# B&R Automation Studio project AutomatedPongGame (part 4)

#### testSet_FieldControl_Idle.c
```c
/********************************************************************
 * COPYRIGHT - MyAutoMation-IT
 ********************************************************************
 * Author: Raivo Berends
 ********************************************************************/

#include <bur/plctypes.h>

#ifdef _DEFAULT_INCLUDES
#include <AsDefault.h>
#endif

#include "UnitTest.h"
#include "Library.h"
#include "CommonTypes.h"
#include <string.h>

_SETUP_TEST(void)
{
	FieldControlFB.FieldControl = &FieldControlStruct;
	FieldControlFB.FieldMotor = &FieldMotorStruct;
	FieldControlFB.InclinoSensor = &InclinoSensorStruct;

	memset(FieldControlFB.FieldControl, 0, sizeof(*FieldControlFB.FieldControl));
	memset(FieldControlFB.FieldMotor, 0, sizeof(*FieldControlFB.FieldMotor));
	memset(FieldControlFB.InclinoSensor, 0, sizeof(*FieldControlFB.InclinoSensor));

	FieldControlFB.FieldControl->STS.StateInt = STATE_IDLE;

	TEST_DONE;
}

_TEST Test_Idle_StaysIdle_WhenNotRunning(void)
{
	FieldControlFB.FieldControl->STS.Running = 0;

	FB_FieldControl(&FieldControlFB);

	TEST_ASSERT_EQUAL_INT(STATE_IDLE, FieldControlFB.FieldControl->STS.StateInt);

	TEST_DONE;
}

_TEST Test_Idle_TransitionsToRunning(void)
{
	FieldControlFB.FieldControl->STS.Running = 1;

	FB_FieldControl(&FieldControlFB);

	TEST_ASSERT_EQUAL_INT(STATE_RUNNING, FieldControlFB.FieldControl->STS.StateInt);

	TEST_DONE;
}

/*
B+R UnitTest: This is generated code.
Do not edit! Do not move!
Description: UnitTest Testprogramm infrastructure (TestSet).
LastUpdated: 2026-05-07 13:23:22Z
By B+R UnitTest Helper Version: 2.0.2.35
*/
UNITTEST_FIXTURES(fixtures)
{
	new_TestFixture("Test_Idle_StaysIdle_WhenNotRunning", Test_Idle_StaysIdle_WhenNotRunning),
	new_TestFixture("Test_Idle_TransitionsToRunning", Test_Idle_TransitionsToRunning),
};

UNITTEST_CALLER_COMPLETE_EXPLICIT(testSet_FieldControl_Idle, "testSet_FieldControl_Idle", setupTest, 0, fixtures, 0, 0, 0);
```

#### testSet_FieldControl_Running.c
```c
/********************************************************************
 * COPYRIGHT - MyAutoMation-IT
 ********************************************************************
 * Author: Raivo Berends
 ********************************************************************/

#include <bur/plctypes.h>

#ifdef _DEFAULT_INCLUDES
#include <AsDefault.h>
#endif

#include "UnitTest.h"
#include "Library.h"
#include "CommonTypes.h"
#include <string.h>

_SETUP_TEST(void)
{
	FieldControlFB.FieldControl = &FieldControlStruct;
	FieldControlFB.FieldMotor = &FieldMotorStruct;
	FieldControlFB.InclinoSensor = &InclinoSensorStruct;

	memset(FieldControlFB.FieldControl, 0, sizeof(*FieldControlFB.FieldControl));
	memset(FieldControlFB.FieldMotor, 0, sizeof(*FieldControlFB.FieldMotor));
	memset(FieldControlFB.InclinoSensor, 0, sizeof(*FieldControlFB.InclinoSensor));

	FieldControlFB.FieldControl->STS.StateInt = STATE_RUNNING;

	TEST_DONE;
}

_TEST Test_Running_ResetsStopCommand(void)
{
	FieldControlFB.FieldMotor->CS.Stop = 1;

	FB_FieldControl(&FieldControlFB);

	TEST_ASSERT_EQUAL_INT(0, FieldControlFB.FieldMotor->CS.Stop);

	TEST_DONE;
}

_TEST Test_Running_DisablesJogNeg_WhenAtMaxAngle(void)
{
	FieldControlFB.FieldControl->STS.CurrentAngle = MAX_ANGLE;

	FieldControlFB.FieldMotor->HMI.MoveJogNeg = 1;

	FB_FieldControl(&FieldControlFB);

	TEST_ASSERT_EQUAL_INT(0, FieldControlFB.FieldMotor->HMI.MoveJogNeg);

	TEST_DONE;
}

_TEST Test_Running_DisablesJogNeg_WhenAboveMaxAngle(void)
{
	FieldControlFB.FieldControl->STS.CurrentAngle = 25.0;

	FieldControlFB.FieldMotor->HMI.MoveJogNeg = 1;

	FB_FieldControl(&FieldControlFB);

	TEST_ASSERT_EQUAL_INT(0, FieldControlFB.FieldMotor->HMI.MoveJogNeg);

	TEST_DONE;
}

_TEST Test_Running_DisablesJogPos_WhenAtMinAngle(void)
{
	FieldControlFB.FieldControl->STS.CurrentAngle = MIN_ANGLE;

	FieldControlFB.FieldMotor->HMI.MoveJogPos = 1;

	FB_FieldControl(&FieldControlFB);

	TEST_ASSERT_EQUAL_INT(0, FieldControlFB.FieldMotor->HMI.MoveJogPos);

	TEST_DONE;
}

_TEST Test_Running_DisablesJogPos_WhenBelowMinAngle(void)
{
	FieldControlFB.FieldControl->STS.CurrentAngle = 0.0;

	FieldControlFB.FieldMotor->HMI.MoveJogPos = 1;

	FB_FieldControl(&FieldControlFB);

	TEST_ASSERT_EQUAL_INT(0, FieldControlFB.FieldMotor->HMI.MoveJogPos);

	TEST_DONE;
}

_TEST Test_Running_DoesNotChangeJogCommands_WithinLimits(void)
{
	FieldControlFB.FieldControl->STS.CurrentAngle = 10.0;

	FieldControlFB.FieldMotor->HMI.MoveJogNeg = 1;
	FieldControlFB.FieldMotor->HMI.MoveJogPos = 1;

	FB_FieldControl(&FieldControlFB);

	TEST_ASSERT_EQUAL_INT(1, FieldControlFB.FieldMotor->HMI.MoveJogNeg);
	TEST_ASSERT_EQUAL_INT(1, FieldControlFB.FieldMotor->HMI.MoveJogPos);

	TEST_DONE;
}

_TEST Test_Running_MaxAngle_DoesNotChangeJogPos(void)
{
	FieldControlFB.FieldControl->STS.CurrentAngle = MAX_ANGLE;

	FieldControlFB.FieldMotor->HMI.MoveJogNeg = 1;
	FieldControlFB.FieldMotor->HMI.MoveJogPos = 1;

	FB_FieldControl(&FieldControlFB);

	TEST_ASSERT_EQUAL_INT(0, FieldControlFB.FieldMotor->HMI.MoveJogNeg);
	TEST_ASSERT_EQUAL_INT(1, FieldControlFB.FieldMotor->HMI.MoveJogPos);

	TEST_DONE;
}
/*
B+R UnitTest: This is generated code.
Do not edit! Do not move!
Description: UnitTest Testprogramm infrastructure (TestSet).
LastUpdated: 2026-05-07 13:23:22Z
By B+R UnitTest Helper Version: 2.0.2.35
*/
UNITTEST_FIXTURES(fixtures)
{
	new_TestFixture("Test_Running_ResetsStopCommand", Test_Running_ResetsStopCommand),
	new_TestFixture("Test_Running_DisablesJogNeg_WhenAtMaxAngle", Test_Running_DisablesJogNeg_WhenAtMaxAngle),
	new_TestFixture("Test_Running_DisablesJogNeg_WhenAboveMaxAngle", Test_Running_DisablesJogNeg_WhenAboveMaxAngle),
	new_TestFixture("Test_Running_DisablesJogPos_WhenAtMinAngle", Test_Running_DisablesJogPos_WhenAtMinAngle),
	new_TestFixture("Test_Running_DisablesJogPos_WhenBelowMinAngle", Test_Running_DisablesJogPos_WhenBelowMinAngle),
	new_TestFixture("Test_Running_DoesNotChangeJogCommands_WithinLimits", Test_Running_DoesNotChangeJogCommands_WithinLimits),
	new_TestFixture("Test_Running_MaxAngle_DoesNotChangeJogPos", Test_Running_MaxAngle_DoesNotChangeJogPos),
};

UNITTEST_CALLER_COMPLETE_EXPLICIT(testSet_FieldControl_Running, "testSet_FieldControl_Running", setupTest, 0, fixtures, 0, 0, 0);
```

#### testSet_FieldControl_Stopping.c
```c
/********************************************************************
 * COPYRIGHT - MyAutoMation-IT
 ********************************************************************
 * Author: Raivo Berends
 ********************************************************************/

#include <bur/plctypes.h>

#ifdef _DEFAULT_INCLUDES
#include <AsDefault.h>
#endif

#include "UnitTest.h"
#include "Library.h"
#include "CommonTypes.h"
#include <string.h>

_SETUP_TEST(void)
{
	FieldControlFB.FieldControl = &FieldControlStruct;
	FieldControlFB.FieldMotor = &FieldMotorStruct;
	FieldControlFB.InclinoSensor = &InclinoSensorStruct;

	memset(FieldControlFB.FieldControl, 0, sizeof(*FieldControlFB.FieldControl));
	memset(FieldControlFB.FieldMotor, 0, sizeof(*FieldControlFB.FieldMotor));
	memset(FieldControlFB.InclinoSensor, 0, sizeof(*FieldControlFB.InclinoSensor));

	FieldControlFB.FieldControl->STS.StateInt = STATE_STOPPING;

	TEST_DONE;
}

_TEST Test_Stopping_StaysStopping_WhenNotDisabled(void)
{
	FieldControlFB.FieldControl->STS.Disabled = 0;

	FB_FieldControl(&FieldControlFB);

	TEST_ASSERT_EQUAL_INT(STATE_STOPPING, FieldControlFB.FieldControl->STS.StateInt);

	TEST_DONE;
}

_TEST Test_Stopping_TransitionsToDisabled(void)
{
	FieldControlFB.FieldControl->STS.Disabled = 1;

	FB_FieldControl(&FieldControlFB);

	TEST_ASSERT_EQUAL_INT(STATE_DISABLED, FieldControlFB.FieldControl->STS.StateInt);

	TEST_DONE;
}
/*
B+R UnitTest: This is generated code.
Do not edit! Do not move!
Description: UnitTest Testprogramm infrastructure (TestSet).
LastUpdated: 2026-05-07 13:23:22Z
By B+R UnitTest Helper Version: 2.0.2.35
*/
UNITTEST_FIXTURES(fixtures)
{
	new_TestFixture("Test_Stopping_StaysStopping_WhenNotDisabled", Test_Stopping_StaysStopping_WhenNotDisabled),
	new_TestFixture("Test_Stopping_TransitionsToDisabled", Test_Stopping_TransitionsToDisabled),
};

UNITTEST_CALLER_COMPLETE_EXPLICIT(testSet_FieldControl_Stopping, "testSet_FieldControl_Stopping", setupTest, 0, fixtures, 0, 0, 0);
```

### Program Logical/UnitTests/UnitTests/Tests_InclinoSensor_C (ANSIC)

#### variables.var - Name the suite and add PVs for the program
```iecst
(********************************************************************
 * COPYRIGHT --  MyAutomation-IT
 ********************************************************************
 * Program: Tests_InclinoSensor_C
 * File: variables.var
 * Author: Raivo Berends
 ********************************************************************
 * Local variables of program Tests_InclinoSensor_C
 ********************************************************************)
(*Describe the test*)
VAR
	Testsuite : UtMgrTestSuite := (Name:='InclinoSensor_Tests',Type:=utMgrTEST_TYPE_C);
END_VAR
(*Variables used in the tests*)
VAR
	InclinoSensorFB : FB_InclinoSensor;
	InclinoSensorStruct : UDT_InclinoSensor;
END_VAR
```

#### autoGeneratedFile.c - Auto generated code - list of all test sets in the program
```c
/*
B+R UnitTest: This is generated code.
Do not edit! Do not move!
Description: UnitTest Testprogramm infrastructure (List of TestSets).
LastUpdated: 2026-05-07 09:44:28Z
By B+R UnitTest Helper Version: 2.0.2.35
*/
#include "UnitTest.h"

UNITTEST_TESTSET_DECLARATION  testSet_InclinoSensor;

UNITTEST_TESTSET_FIXTURES(utTestSets)
{
	new_TestSet(testSet_InclinoSensor),
};
UNTITTEST_TESTSET_HANDLER();
```

#### testSet_InclinoSensor.c
```c
/********************************************************************
 * COPYRIGHT - MyAutoMation-IT
 ********************************************************************
 * Author: Raivo Berends
 ********************************************************************/

#include <bur/plctypes.h>

#ifdef _DEFAULT_INCLUDES
#include <AsDefault.h>
#endif

#include "UnitTest.h"
#include "Library.h"
#include "CommonTypes.h"
#include <string.h>

_SETUP_TEST(void)
{
	InclinoSensorFB.InclinoSensor = &InclinoSensorStruct;
	memset(	InclinoSensorFB.InclinoSensor, 0, sizeof(*InclinoSensorFB.InclinoSensor));

	TEST_DONE;
}

_TEST Test_InclinoSensor_CalculatesAngleFromRawData(void)
{
	InclinoSensorFB.InclinoSensor->IO.DataMSB = 0x01;
	InclinoSensorFB.InclinoSensor->IO.DataLSB = 0x00;

	FB_InclinoSensor(&InclinoSensorFB);

	TEST_ASSERT_EQUAL_FLOAT((float)256 / TO_DEGREES, InclinoSensorFB.InclinoSensor->STS.CurrentAngle);

	TEST_DONE;
}

_TEST Test_InclinoSensor_CalculatesNegativeAngle(void)
{
	InclinoSensorFB.InclinoSensor->IO.DataMSB = 0xFF;
	InclinoSensorFB.InclinoSensor->IO.DataLSB = 0x00;

	FB_InclinoSensor(&InclinoSensorFB);

	TEST_ASSERT_EQUAL_FLOAT((float)((INT)((0xFF00))) / TO_DEGREES, InclinoSensorFB.InclinoSensor->STS.CurrentAngle);

	TEST_DONE;
}

_TEST Test_InclinoSensor_SetsAlarmColourGreen(void)
{
	InclinoSensorFB.InclinoSensor->STS.AlarmActive = 0;

	FB_InclinoSensor(&InclinoSensorFB);

	TEST_ASSERT_EQUAL_INT(GREEN_COLOUR, InclinoSensorFB.InclinoSensor->STS.AlarmActiveColour);

	TEST_DONE;
}

_TEST Test_InclinoSensor_SetsAlarmColourRed(void)
{
	InclinoSensorFB.InclinoSensor->STS.AlarmActive = 1;

	FB_InclinoSensor(&InclinoSensorFB);

	TEST_ASSERT_EQUAL_INT(RED_COLOUR, InclinoSensorFB.InclinoSensor->STS.AlarmActiveColour);

	TEST_DONE;
}

_TEST Test_InclinoSensor_SetCenterPoint_NormalMode(void)
{
	InclinoSensorFB.InclinoSensor->CS.SetCenterPoint = 0;

	FB_InclinoSensor(&InclinoSensorFB);

	TEST_ASSERT_EQUAL_INT(CENTERPOINT_NORMAL, InclinoSensorFB.InclinoSensor->IO.SetCenterPoint);

	TEST_DONE;
}

_TEST Test_InclinoSensor_SetCenterPoint_CalibrationMode(void)
{
	InclinoSensorFB.InclinoSensor->CS.SetCenterPoint = 1;

	FB_InclinoSensor(&InclinoSensorFB);

	TEST_ASSERT_EQUAL_INT(CENTERPOINT_SET, InclinoSensorFB.InclinoSensor->IO.SetCenterPoint);

	TEST_DONE;
}

_TEST Test_InclinoSensor_RawBitCombination(void)
{
	InclinoSensorFB.InclinoSensor->IO.DataMSB = 0x12;
	InclinoSensorFB.InclinoSensor->IO.DataLSB = 0x34;

	FB_InclinoSensor(&InclinoSensorFB);

	TEST_ASSERT_EQUAL_INT((0x1234), (INT)((InclinoSensorFB.InclinoSensor->STS.CurrentAngle * TO_DEGREES) + 1));

	TEST_DONE;
}

/*
B+R UnitTest: This is generated code.
Do not edit! Do not move!
Description: UnitTest Testprogramm infrastructure (TestSet).
LastUpdated: 2026-05-07 09:44:28Z
By B+R UnitTest Helper Version: 2.0.2.35
*/
UNITTEST_FIXTURES(fixtures)
{
	new_TestFixture("Test_InclinoSensor_CalculatesAngleFromRawData", Test_InclinoSensor_CalculatesAngleFromRawData),
	new_TestFixture("Test_InclinoSensor_CalculatesNegativeAngle", Test_InclinoSensor_CalculatesNegativeAngle),
	new_TestFixture("Test_InclinoSensor_SetsAlarmColourGreen", Test_InclinoSensor_SetsAlarmColourGreen),
	new_TestFixture("Test_InclinoSensor_SetsAlarmColourRed", Test_InclinoSensor_SetsAlarmColourRed),
	new_TestFixture("Test_InclinoSensor_SetCenterPoint_NormalMode", Test_InclinoSensor_SetCenterPoint_NormalMode),
	new_TestFixture("Test_InclinoSensor_SetCenterPoint_CalibrationMode", Test_InclinoSensor_SetCenterPoint_CalibrationMode),
	new_TestFixture("Test_InclinoSensor_RawBitCombination", Test_InclinoSensor_RawBitCombination),
};

UNITTEST_CALLER_COMPLETE_EXPLICIT(testSet_InclinoSensor, "testSet_InclinoSensor", setupTest, 0, fixtures, 0, 0, 0);
```

### Program Logical/UnitTests/UnitTests/Tests_PongGame_C (ANSIC)

#### variables.var - Name the suite and add PVs for the program
```iecst
(********************************************************************
 * COPYRIGHT --  MyAutomation-IT
 ********************************************************************
 * Program: Tests_PongGame_C
 * File: variables.var
 * Author: Raivo Berends
 ********************************************************************
 * Local variables of program Tests_PongGame_C
 ********************************************************************)
(*Describe the test*)
VAR
	Testsuite : UtMgrTestSuite := (Name:='PongGame_Tests',Type:=utMgrTEST_TYPE_C);
END_VAR
(*Variables used in the tests*)
VAR
	PongGameFB : FB_PongGame;
	PongGameStruct : UDT_PongGame;
	BallControlStruct : UDT_BallControl;
	FieldControlStruct : UDT_FieldControl;
END_VAR
```

#### autoGeneratedFile.c - Auto generated code - list of all test sets in the program
```c
/*
B+R UnitTest: This is generated code.
Do not edit! Do not move!
Description: UnitTest Testprogramm infrastructure (List of TestSets).
LastUpdated: 2026-05-07 13:54:36Z
By B+R UnitTest Helper Version: 2.0.2.35
*/
#include "UnitTest.h"

UNITTEST_TESTSET_DECLARATION  testSet_PongGame_Disabled;
UNITTEST_TESTSET_DECLARATION  testSet_PongGame_Initializing;
UNITTEST_TESTSET_DECLARATION  testSet_PongGame_Idle;
UNITTEST_TESTSET_DECLARATION  testSet_PongGame_Running;
UNITTEST_TESTSET_DECLARATION  testSet_PongGame_Stopping;

UNITTEST_TESTSET_FIXTURES(utTestSets)
{
	new_TestSet(testSet_PongGame_Disabled),
	new_TestSet(testSet_PongGame_Initializing),
	new_TestSet(testSet_PongGame_Idle),
	new_TestSet(testSet_PongGame_Running),
	new_TestSet(testSet_PongGame_Stopping),
};
UNTITTEST_TESTSET_HANDLER();
```

#### testSet_PongGame_Disabled.c
```c
/********************************************************************
 * COPYRIGHT - MyAutoMation-IT
 ********************************************************************
 * Author: Raivo Berends
 ********************************************************************/

#include <bur/plctypes.h>

#ifdef _DEFAULT_INCLUDES
#include <AsDefault.h>
#endif

#include "UnitTest.h"
#include "Library.h"
#include "CommonTypes.h"
#include <string.h>

_SETUP_TEST(void)
{
	PongGameFB.PongGame = &PongGameStruct;
	PongGameFB.BallControl = &BallControlStruct;
	PongGameFB.FieldControl = &FieldControlStruct;

	memset(PongGameFB.PongGame, 0, sizeof(*PongGameFB.PongGame));
	memset(PongGameFB.BallControl, 0, sizeof(*PongGameFB.BallControl));
	memset(PongGameFB.FieldControl, 0, sizeof(*PongGameFB.FieldControl));

	PongGameFB.PongGame->STS.StateInt = STATE_DISABLED;

	TEST_DONE;
}

_TEST Test_Disabled_ResetsRuntimeValues(void)
{
	PongGameFB.PongGame->CS.StopGame = 0;
	PongGameFB.PongGame->HMI.StopGame = 0;

	PongGameFB.PongGame->STS.GameStopped = 1;

	FB_PongGame(&PongGameFB);

	TEST_ASSERT_EQUAL_INT(0, PongGameFB.PongGame->STS.GameStopped);
	TEST_ASSERT_EQUAL_INT(0, PongGameFB.PongGame->CS.StopGame);

	TEST_DONE;
}

_TEST Test_Disabled_SetsStateString(void)
{
	PongGameFB.PongGame->CS.StopGame = 0;
	PongGameFB.PongGame->HMI.StopGame = 0;

	FB_PongGame(&PongGameFB);

	TEST_ASSERT_EQUAL_STRING("Disabled", PongGameFB.PongGame->STS.StateString);

	TEST_DONE;
}

_TEST Test_Disabled_TransitionsToInitializing(void)
{
	PongGameFB.PongGame->CS.StopGame = 0;
	PongGameFB.PongGame->HMI.StopGame = 0;

	PongGameFB.PongGame->STS.Initializing = 1;

	FB_PongGame(&PongGameFB);

	TEST_ASSERT_EQUAL_INT(STATE_INITIALIZING, PongGameFB.PongGame->STS.StateInt);

	TEST_DONE;
}

_TEST Test_Disabled_StaysDisabled_WhenNotInitializing(void)
{
	PongGameFB.PongGame->CS.StopGame = 0;
	PongGameFB.PongGame->HMI.StopGame = 0;

	PongGameFB.PongGame->STS.Initializing = 0;

	FB_PongGame(&PongGameFB);

	TEST_ASSERT_EQUAL_INT(STATE_DISABLED, PongGameFB.PongGame->STS.StateInt);

	TEST_DONE;
}

_TEST Test_Disabled_OverwriteExistingValues(void)
{
	PongGameFB.PongGame->CS.StopGame = 0;
	PongGameFB.PongGame->HMI.StopGame = 0;

	PongGameFB.PongGame->STS.GameStopped = 1;

	FB_PongGame(&PongGameFB);

	TEST_ASSERT_EQUAL_INT(0, PongGameFB.PongGame->STS.GameStopped);
	TEST_ASSERT_EQUAL_INT(0, PongGameFB.PongGame->CS.StopGame);

	TEST_DONE;
}

_TEST Test_Disabled_StillResetsValues_BeforeInitializingTransition(void)
{
	PongGameFB.PongGame->CS.StopGame = 0;
	PongGameFB.PongGame->HMI.StopGame = 0;

	PongGameFB.PongGame->STS.GameStopped = 1;

	PongGameFB.PongGame->STS.Initializing = 1;

	FB_PongGame(&PongGameFB);

	TEST_ASSERT_EQUAL_INT(0, PongGameFB.PongGame->STS.GameStopped);
	TEST_ASSERT_EQUAL_INT(0, PongGameFB.PongGame->CS.StopGame);

	TEST_ASSERT_EQUAL_INT(STATE_INITIALIZING, PongGameFB.PongGame->STS.StateInt);

	TEST_DONE;
}

_TEST Test_Disabled_StopGame_TransitionsToStopping(void)
{
	PongGameFB.PongGame->CS.StopGame = 1;

	PongGameFB.PongGame->STS.AlarmActive = 0;
	PongGameFB.PongGame->STS.Interlocked = 0;

	FB_PongGame(&PongGameFB);

	TEST_ASSERT_EQUAL_INT(STATE_STOPPING, PongGameFB.PongGame->STS.StateInt);

	TEST_DONE;
}

_TEST Test_Disabled_HMIStopGame_TransitionsToStopping(void)
{
	PongGameFB.PongGame->HMI.StopGame = 1;

	PongGameFB.PongGame->STS.AlarmActive = 0;
	PongGameFB.PongGame->STS.Interlocked = 0;

	FB_PongGame(&PongGameFB);

	TEST_ASSERT_EQUAL_INT(STATE_STOPPING, PongGameFB.PongGame->STS.StateInt);

	TEST_DONE;
}

_TEST Test_Disabled_StopGameBlockedByInterlock(void)
{
	PongGameFB.PongGame->CS.StopGame = 1;

	PongGameFB.PongGame->STS.AlarmActive = 0;
	PongGameFB.PongGame->STS.Interlocked = 1;

	FB_PongGame(&PongGameFB);

	TEST_ASSERT_EQUAL_INT(STATE_DISABLED, PongGameFB.PongGame->STS.StateInt);

	TEST_DONE;
}
/*
B+R UnitTest: This is generated code.
Do not edit! Do not move!
Description: UnitTest Testprogramm infrastructure (TestSet).
LastUpdated: 2026-05-08 07:49:02Z
By B+R UnitTest Helper Version: 2.0.2.35
*/
UNITTEST_FIXTURES(fixtures)
{
	new_TestFixture("Test_Disabled_ResetsRuntimeValues", Test_Disabled_ResetsRuntimeValues),
	new_TestFixture("Test_Disabled_SetsStateString", Test_Disabled_SetsStateString),
	new_TestFixture("Test_Disabled_TransitionsToInitializing", Test_Disabled_TransitionsToInitializing),
	new_TestFixture("Test_Disabled_StaysDisabled_WhenNotInitializing", Test_Disabled_StaysDisabled_WhenNotInitializing),
	new_TestFixture("Test_Disabled_OverwriteExistingValues", Test_Disabled_OverwriteExistingValues),
	new_TestFixture("Test_Disabled_StillResetsValues_BeforeInitializingTransition", Test_Disabled_StillResetsValues_BeforeInitializingTransition),
	new_TestFixture("Test_Disabled_StopGame_TransitionsToStopping", Test_Disabled_StopGame_TransitionsToStopping),
	new_TestFixture("Test_Disabled_HMIStopGame_TransitionsToStopping", Test_Disabled_HMIStopGame_TransitionsToStopping),
	new_TestFixture("Test_Disabled_StopGameBlockedByInterlock", Test_Disabled_StopGameBlockedByInterlock),
};

UNITTEST_CALLER_COMPLETE_EXPLICIT(testSet_PongGame_Disabled, "testSet_PongGame_Disabled", setupTest, 0, fixtures, 0, 0, 0);
```

#### testSet_PongGame_Initializing.c
```c
/********************************************************************
 * COPYRIGHT - MyAutoMation-IT
 ********************************************************************
 * Author: Raivo Berends
 ********************************************************************/

#include <bur/plctypes.h>

#ifdef _DEFAULT_INCLUDES
#include <AsDefault.h>
#endif

#include "UnitTest.h"
#include "Library.h"
#include "CommonTypes.h"
#include <string.h>

_SETUP_TEST(void)
{
	PongGameFB.PongGame = &PongGameStruct;
	PongGameFB.BallControl = &BallControlStruct;
	PongGameFB.FieldControl = &FieldControlStruct;

	memset(PongGameFB.PongGame, 0, sizeof(*PongGameFB.PongGame));
	memset(PongGameFB.BallControl, 0, sizeof(*PongGameFB.BallControl));
	memset(PongGameFB.FieldControl, 0, sizeof(*PongGameFB.FieldControl));

	PongGameFB.PongGame->STS.StateInt = STATE_INITIALIZING;

	TEST_DONE;
}

_TEST Test_Initializing_SetsStateString(void)
{
	PongGameFB.PongGame->STS.Idle = 0;

	FB_PongGame(&PongGameFB);

	TEST_ASSERT_EQUAL_STRING("Initializing...", PongGameFB.PongGame->STS.StateString);

	TEST_DONE;
}

_TEST Test_Initializing_StaysWhenNotIdle(void)
{
	PongGameFB.PongGame->STS.Idle = 0;

	FB_PongGame(&PongGameFB);

	TEST_ASSERT_EQUAL_INT(STATE_INITIALIZING, PongGameFB.PongGame->STS.StateInt);

	TEST_DONE;
}

_TEST Test_Initializing_TransitionsToIdle(void)
{
	PongGameFB.PongGame->STS.Idle = 1;

	FB_PongGame(&PongGameFB);

	TEST_ASSERT_EQUAL_INT(STATE_IDLE, PongGameFB.PongGame->STS.StateInt);

	TEST_DONE;
}

_TEST Test_Initializing_IdleHasPriority(void)
{
	PongGameFB.PongGame->STS.Idle = 1;

	FB_PongGame(&PongGameFB);

	TEST_ASSERT_EQUAL_INT(STATE_IDLE, PongGameFB.PongGame->STS.StateInt);
	TEST_ASSERT_EQUAL_STRING("Initializing...", PongGameFB.PongGame->STS.StateString);

	TEST_DONE;
}

_TEST Test_Initializing_ResetScore(void)
{
	PongGameFB.PongGame->PAR.Score = 99;

	FB_PongGame(&PongGameFB);

	TEST_ASSERT_EQUAL_INT(0, PongGameFB.PongGame->PAR.Score);

	TEST_DONE;
}

/*
B+R UnitTest: This is generated code.
Do not edit! Do not move!
Description: UnitTest Testprogramm infrastructure (TestSet).
LastUpdated: 2026-05-19 08:38:02Z
By B+R UnitTest Helper Version: 2.0.2.35
*/
UNITTEST_FIXTURES(fixtures)
{
	new_TestFixture("Test_Initializing_SetsStateString", Test_Initializing_SetsStateString),
	new_TestFixture("Test_Initializing_StaysWhenNotIdle", Test_Initializing_StaysWhenNotIdle),
	new_TestFixture("Test_Initializing_TransitionsToIdle", Test_Initializing_TransitionsToIdle),
	new_TestFixture("Test_Initializing_IdleHasPriority", Test_Initializing_IdleHasPriority),
	new_TestFixture("Test_Initializing_ResetScore", Test_Initializing_ResetScore),
};

UNITTEST_CALLER_COMPLETE_EXPLICIT(testSet_PongGame_Initializing, "testSet_PongGame_Initializing", setupTest, 0, fixtures, 0, 0, 0);
```

#### testSet_PongGame_Idle.c
```c
/********************************************************************
 * COPYRIGHT - MyAutoMation-IT
 ********************************************************************
 * Author: Raivo Berends
 ********************************************************************/

#include <bur/plctypes.h>

#ifdef _DEFAULT_INCLUDES
#include <AsDefault.h>
#endif

#include "UnitTest.h"
#include "Library.h"
#include "CommonTypes.h"
#include <string.h>

_SETUP_TEST(void)
{
	PongGameFB.PongGame = &PongGameStruct;
	PongGameFB.BallControl = &BallControlStruct;
	PongGameFB.FieldControl = &FieldControlStruct;

	memset(PongGameFB.PongGame, 0, sizeof(*PongGameFB.PongGame));
	memset(PongGameFB.BallControl, 0, sizeof(*PongGameFB.BallControl));
	memset(PongGameFB.FieldControl, 0, sizeof(*PongGameFB.FieldControl));

	PongGameFB.PongGame->STS.StateInt = STATE_IDLE;

	TEST_DONE;
}

_TEST Test_Idle_SetsStateString(void)
{
	PongGameFB.PongGame->STS.Running = 0;

	FB_PongGame(&PongGameFB);

	TEST_ASSERT_EQUAL_STRING("Idle", PongGameFB.PongGame->STS.StateString);

	TEST_DONE;
}

_TEST Test_Idle_StaysIdle_WhenNotRunning(void)
{
	PongGameFB.PongGame->STS.Running = 0;

	FB_PongGame(&PongGameFB);

	TEST_ASSERT_EQUAL_INT(STATE_IDLE, PongGameFB.PongGame->STS.StateInt);

	TEST_DONE;
}

_TEST Test_Idle_TransitionsToRunning(void)
{
	PongGameFB.PongGame->STS.Running = 1;

	FB_PongGame(&PongGameFB);

	TEST_ASSERT_EQUAL_INT(STATE_RUNNING, PongGameFB.PongGame->STS.StateInt);

	TEST_DONE;
}

_TEST Test_Idle_RunningOverridesIdleState(void)
{
	PongGameFB.PongGame->STS.Running = 1;

	FB_PongGame(&PongGameFB);

	TEST_ASSERT_EQUAL_INT(STATE_RUNNING, PongGameFB.PongGame->STS.StateInt);

	TEST_ASSERT_EQUAL_STRING("Idle", PongGameFB.PongGame->STS.StateString);

	TEST_DONE;
}
/*
B+R UnitTest: This is generated code.
Do not edit! Do not move!
Description: UnitTest Testprogramm infrastructure (TestSet).
LastUpdated: 2026-05-07 13:59:14Z
By B+R UnitTest Helper Version: 2.0.2.35
*/
UNITTEST_FIXTURES(fixtures)
{
	new_TestFixture("Test_Idle_SetsStateString", Test_Idle_SetsStateString),
	new_TestFixture("Test_Idle_StaysIdle_WhenNotRunning", Test_Idle_StaysIdle_WhenNotRunning),
	new_TestFixture("Test_Idle_TransitionsToRunning", Test_Idle_TransitionsToRunning),
	new_TestFixture("Test_Idle_RunningOverridesIdleState", Test_Idle_RunningOverridesIdleState),
};

UNITTEST_CALLER_COMPLETE_EXPLICIT(testSet_PongGame_Idle, "testSet_PongGame_Idle", setupTest, 0, fixtures, 0, 0, 0);
```

#### testSet_PongGame_Running.c
```c
/********************************************************************
 * COPYRIGHT - MyAutoMation-IT
 ********************************************************************
 * Author: Raivo Berends
 ********************************************************************/

#include <bur/plctypes.h>

#ifdef _DEFAULT_INCLUDES
#include <AsDefault.h>
#endif

#include "UnitTest.h"
#include "Library.h"
#include "CommonTypes.h"
#include <string.h>

_SETUP_TEST(void)
{
	PongGameFB.PongGame = &PongGameStruct;
	PongGameFB.BallControl = &BallControlStruct;
	PongGameFB.FieldControl = &FieldControlStruct;

	memset(PongGameFB.PongGame, 0, sizeof(*PongGameFB.PongGame));
	memset(PongGameFB.BallControl, 0, sizeof(*PongGameFB.BallControl));
	memset(PongGameFB.FieldControl, 0, sizeof(*PongGameFB.FieldControl));

	PongGameFB.PongGame->STS.StateInt = STATE_RUNNING;

	TEST_DONE;
}

_TEST Test_Running_SetsStateString(void)
{
	PongGameFB.BallControl->STS.ShootCycleCompleted = 0;
	PongGameFB.BallControl->STS.GameOver = 0;

	FB_PongGame(&PongGameFB);

	TEST_ASSERT_EQUAL_STRING("Running", PongGameFB.PongGame->STS.StateString);

	TEST_DONE;
}

_TEST Test_Running_IncrementsScore_OnShootCycleCompleted(void)
{
	PongGameFB.PongGame->PAR.Score = 10;

	PongGameFB.BallControl->STS.ShootCycleCompleted = 1;
	PongGameFB.BallControl->STS.GameOver = 0;

	FB_PongGame(&PongGameFB);

	TEST_ASSERT_EQUAL_INT(11, PongGameFB.PongGame->PAR.Score);

	TEST_DONE;
}

_TEST Test_Running_DoesNotIncrementScore_WhenNoCycleCompleted(void)
{
	PongGameFB.PongGame->PAR.Score = 10;

	PongGameFB.BallControl->STS.ShootCycleCompleted = 0;
	PongGameFB.BallControl->STS.GameOver = 0;

	FB_PongGame(&PongGameFB);

	TEST_ASSERT_EQUAL_INT(10, PongGameFB.PongGame->PAR.Score);

	TEST_DONE;
}

_TEST Test_Running_GameOver_SetsStopGame(void)
{
	PongGameFB.BallControl->STS.GameOver = 1;
	PongGameFB.BallControl->STS.ShootCycleCompleted = 0;

	FB_PongGame(&PongGameFB);

	TEST_ASSERT_EQUAL_INT(1, PongGameFB.PongGame->CS.StopGame);

	TEST_DONE;
}

_TEST Test_Running_NoGameOver_DoesNotStopGame(void)
{
	PongGameFB.PongGame->CS.StopGame = 0;

	PongGameFB.BallControl->STS.GameOver = 0;
	PongGameFB.BallControl->STS.ShootCycleCompleted = 0;

	FB_PongGame(&PongGameFB);

	TEST_ASSERT_EQUAL_INT(0, PongGameFB.PongGame->CS.StopGame);

	TEST_DONE;
}

_TEST Test_Running_BothEvents_ScoreAndStop(void)
{
	PongGameFB.PongGame->PAR.Score = 5;
	PongGameFB.PongGame->CS.StopGame = 0;

	PongGameFB.BallControl->STS.ShootCycleCompleted = 1;
	PongGameFB.BallControl->STS.GameOver = 1;

	FB_PongGame(&PongGameFB);

	TEST_ASSERT_EQUAL_INT(6, PongGameFB.PongGame->PAR.Score);
	TEST_ASSERT_EQUAL_INT(1, PongGameFB.PongGame->CS.StopGame);

	TEST_DONE;
}

_TEST Test_Running_StopGame_TransitionsToStopping(void)
{
	PongGameFB.PongGame->CS.StopGame = 1;
	PongGameFB.PongGame->STS.AlarmActive = 0;
	PongGameFB.PongGame->STS.Interlocked = 0;

	FB_PongGame(&PongGameFB);

	TEST_ASSERT_EQUAL_INT(STATE_STOPPING, PongGameFB.PongGame->STS.StateInt);

	TEST_DONE;
}

_TEST Test_Running_StopGame_CS_TransitionsToStopping(void)
{
	PongGameFB.PongGame->CS.StopGame = 1;
	PongGameFB.PongGame->STS.AlarmActive = 0;
	PongGameFB.PongGame->STS.Interlocked = 0;

	FB_PongGame(&PongGameFB);

	TEST_ASSERT_EQUAL_INT(STATE_STOPPING, PongGameFB.PongGame->STS.StateInt);

	TEST_DONE;
}

_TEST Test_Running_StopGame_HMI_TransitionsToStopping(void)
{
	PongGameFB.PongGame->HMI.StopGame = 1;
	PongGameFB.PongGame->STS.AlarmActive = 0;
	PongGameFB.PongGame->STS.Interlocked = 0;

	FB_PongGame(&PongGameFB);

	TEST_ASSERT_EQUAL_INT(STATE_STOPPING, PongGameFB.PongGame->STS.StateInt);

	TEST_DONE;
}

_TEST Test_Running_StopGame_BlockedByInterlock(void)
{
	PongGameFB.PongGame->CS.StopGame = 1;
	PongGameFB.PongGame->STS.AlarmActive = 0;
	PongGameFB.PongGame->STS.Interlocked = 1;

	FB_PongGame(&PongGameFB);

	TEST_ASSERT_EQUAL_INT(STATE_RUNNING, PongGameFB.PongGame->STS.StateInt);

	TEST_DONE;
}

_TEST Test_Running_XOR_Start_Command(void)
{
	PongGameFB.PongGame->HMI.Start = 1;
	PongGameFB.PongGame->CS.Start = 1;

	FB_PongGame(&PongGameFB);

	TEST_ASSERT_EQUAL_INT(0, PongGameFB.BallControl->CS.Start);
	TEST_ASSERT_EQUAL_INT(0, PongGameFB.FieldControl->CS.Start);

	TEST_DONE;
}

_TEST Test_Running_XOR_Start_HMI_Only(void)
{
	PongGameFB.PongGame->HMI.Start = 1;
	PongGameFB.PongGame->CS.Start = 0;

	FB_PongGame(&PongGameFB);

	TEST_ASSERT_EQUAL_INT(1, PongGameFB.BallControl->CS.Start);
	TEST_ASSERT_EQUAL_INT(1, PongGameFB.FieldControl->CS.Start);

	TEST_DONE;
}

_TEST Test_Running_XOR_StopGame_Conflict(void)
{
	PongGameFB.PongGame->HMI.StopGame = 1;
	PongGameFB.PongGame->CS.StopGame = 1;

	FB_PongGame(&PongGameFB);

	TEST_ASSERT_EQUAL_INT(0, PongGameFB.BallControl->CS.StopGame);
	TEST_ASSERT_EQUAL_INT(0, PongGameFB.FieldControl->CS.StopGame);

	TEST_DONE;
}

_TEST Test_Running_SubsystemMapping_True(void)
{
	PongGameFB.BallControl->STS.Running = 1;
	PongGameFB.FieldControl->STS.Running = 1;

	FB_PongGame(&PongGameFB);

	TEST_ASSERT_EQUAL_INT(1, PongGameFB.PongGame->STS.Running);

	TEST_DONE;
}

_TEST Test_Running_SubsystemMapping_False(void)
{
	PongGameFB.BallControl->STS.Running = 1;
	PongGameFB.FieldControl->STS.Running = 0;

	FB_PongGame(&PongGameFB);

	TEST_ASSERT_EQUAL_INT(0, PongGameFB.PongGame->STS.Running);

	TEST_DONE;
}

_TEST Test_Running_Interlock_Propagation(void)
{
	PongGameFB.BallControl->STS.Interlocked = 1;
	PongGameFB.FieldControl->STS.Interlocked = 0;

	FB_PongGame(&PongGameFB);

	TEST_ASSERT_EQUAL_INT(1, PongGameFB.PongGame->STS.Interlocked);

	TEST_DONE;
}
/*
B+R UnitTest: This is generated code.
Do not edit! Do not move!
Description: UnitTest Testprogramm infrastructure (TestSet).
LastUpdated: 2026-05-08 07:49:02Z
By B+R UnitTest Helper Version: 2.0.2.35
*/
UNITTEST_FIXTURES(fixtures)
{
	new_TestFixture("Test_Running_SetsStateString", Test_Running_SetsStateString),
	new_TestFixture("Test_Running_IncrementsScore_OnShootCycleCompleted", Test_Running_IncrementsScore_OnShootCycleCompleted),
	new_TestFixture("Test_Running_DoesNotIncrementScore_WhenNoCycleCompleted", Test_Running_DoesNotIncrementScore_WhenNoCycleCompleted),
	new_TestFixture("Test_Running_GameOver_SetsStopGame", Test_Running_GameOver_SetsStopGame),
	new_TestFixture("Test_Running_NoGameOver_DoesNotStopGame", Test_Running_NoGameOver_DoesNotStopGame),
	new_TestFixture("Test_Running_BothEvents_ScoreAndStop", Test_Running_BothEvents_ScoreAndStop),
	new_TestFixture("Test_Running_StopGame_TransitionsToStopping", Test_Running_StopGame_TransitionsToStopping),
	new_TestFixture("Test_Running_StopGame_CS_TransitionsToStopping", Test_Running_StopGame_CS_TransitionsToStopping),
	new_TestFixture("Test_Running_StopGame_HMI_TransitionsToStopping", Test_Running_StopGame_HMI_TransitionsToStopping),
	new_TestFixture("Test_Running_StopGame_BlockedByInterlock", Test_Running_StopGame_BlockedByInterlock),
	new_TestFixture("Test_Running_XOR_Start_Command", Test_Running_XOR_Start_Command),
	new_TestFixture("Test_Running_XOR_Start_HMI_Only", Test_Running_XOR_Start_HMI_Only),
	new_TestFixture("Test_Running_XOR_StopGame_Conflict", Test_Running_XOR_StopGame_Conflict),
	new_TestFixture("Test_Running_SubsystemMapping_True", Test_Running_SubsystemMapping_True),
	new_TestFixture("Test_Running_SubsystemMapping_False", Test_Running_SubsystemMapping_False),
	new_TestFixture("Test_Running_Interlock_Propagation", Test_Running_Interlock_Propagation),
};

UNITTEST_CALLER_COMPLETE_EXPLICIT(testSet_PongGame_Running, "testSet_PongGame_Running", setupTest, 0, fixtures, 0, 0, 0);
```

#### testSet_PongGame_Stopping.c
```c
/********************************************************************
 * COPYRIGHT - MyAutoMation-IT
 ********************************************************************
 * Author: Raivo Berends
 ********************************************************************/

#include <bur/plctypes.h>

#ifdef _DEFAULT_INCLUDES
#include <AsDefault.h>
#endif

#include "UnitTest.h"
#include "Library.h"
#include "CommonTypes.h"
#include <string.h>

_SETUP_TEST(void)
{
	PongGameFB.PongGame = &PongGameStruct;
	PongGameFB.BallControl = &BallControlStruct;
	PongGameFB.FieldControl = &FieldControlStruct;

	memset(PongGameFB.PongGame, 0, sizeof(*PongGameFB.PongGame));
	memset(PongGameFB.BallControl, 0, sizeof(*PongGameFB.BallControl));
	memset(PongGameFB.FieldControl, 0, sizeof(*PongGameFB.FieldControl));

	PongGameFB.PongGame->STS.StateInt = STATE_STOPPING;

	TEST_DONE;
}

_TEST Test_Stopping_ResetsStopGame(void)
{
	PongGameFB.PongGame->CS.StopGame = 1;

	FB_PongGame(&PongGameFB);

	TEST_ASSERT_EQUAL_INT(0, PongGameFB.PongGame->CS.StopGame);

	TEST_DONE;
}

_TEST Test_Stopping_SetsStateString(void)
{
	FB_PongGame(&PongGameFB);

	TEST_ASSERT_EQUAL_STRING("Stopping...", PongGameFB.PongGame->STS.StateString);

	TEST_DONE;
}

_TEST Test_Stopping_UpdatesHighscore_WhenScoreHigher(void)
{
	PongGameFB.PongGame->PAR.Score = 10;
	PongGameFB.PongGame->PAR.Highscore = 5;

	FB_PongGame(&PongGameFB);

	TEST_ASSERT_EQUAL_INT(10, PongGameFB.PongGame->PAR.Highscore);

	TEST_DONE;
}

_TEST Test_Stopping_DoesNotUpdateHighscore_WhenScoreLower(void)
{
	PongGameFB.PongGame->PAR.Score = 5;
	PongGameFB.PongGame->PAR.Highscore = 10;

	FB_PongGame(&PongGameFB);

	TEST_ASSERT_EQUAL_INT(10, PongGameFB.PongGame->PAR.Highscore);

	TEST_DONE;
}

_TEST Test_Stopping_TransitionsToDisabled(void)
{
	PongGameFB.PongGame->STS.Disabled = 1;

	FB_PongGame(&PongGameFB);

	TEST_ASSERT_EQUAL_INT(STATE_DISABLED, PongGameFB.PongGame->STS.StateInt);

	TEST_DONE;
}

_TEST Test_Stopping_StaysStopping_WhenNotDisabled(void)
{
	PongGameFB.PongGame->STS.Disabled = 0;

	FB_PongGame(&PongGameFB);

	TEST_ASSERT_EQUAL_INT(STATE_STOPPING, PongGameFB.PongGame->STS.StateInt);

	TEST_DONE;
}

_TEST Test_Stopping_FullFlow_UpdateAndTransition(void)
{
	PongGameFB.PongGame->CS.StopGame = 1;
	PongGameFB.PongGame->PAR.Score = 12;
	PongGameFB.PongGame->PAR.Highscore = 10;

	PongGameFB.PongGame->STS.Disabled = 1;

	FB_PongGame(&PongGameFB);

	TEST_ASSERT_EQUAL_INT(0, PongGameFB.PongGame->CS.StopGame);
	TEST_ASSERT_EQUAL_INT(12, PongGameFB.PongGame->PAR.Highscore);
	TEST_ASSERT_EQUAL_INT(STATE_DISABLED, PongGameFB.PongGame->STS.StateInt);

	TEST_DONE;
}
/*
B+R UnitTest: This is generated code.
Do not edit! Do not move!
Description: UnitTest Testprogramm infrastructure (TestSet).
LastUpdated: 2026-05-07 13:59:14Z
By B+R UnitTest Helper Version: 2.0.2.35
*/
UNITTEST_FIXTURES(fixtures)
{
	new_TestFixture("Test_Stopping_ResetsStopGame", Test_Stopping_ResetsStopGame),
	new_TestFixture("Test_Stopping_SetsStateString", Test_Stopping_SetsStateString),
	new_TestFixture("Test_Stopping_UpdatesHighscore_WhenScoreHigher", Test_Stopping_UpdatesHighscore_WhenScoreHigher),
	new_TestFixture("Test_Stopping_DoesNotUpdateHighscore_WhenScoreLower", Test_Stopping_DoesNotUpdateHighscore_WhenScoreLower),
	new_TestFixture("Test_Stopping_TransitionsToDisabled", Test_Stopping_TransitionsToDisabled),
	new_TestFixture("Test_Stopping_StaysStopping_WhenNotDisabled", Test_Stopping_StaysStopping_WhenNotDisabled),
	new_TestFixture("Test_Stopping_FullFlow_UpdateAndTransition", Test_Stopping_FullFlow_UpdateAndTransition),
};

UNITTEST_CALLER_COMPLETE_EXPLICIT(testSet_PongGame_Stopping, "testSet_PongGame_Stopping", setupTest, 0, fixtures, 0, 0, 0);
```

### Program Logical/UnitTests/UnitTests/Tests_Shooter_C (ANSIC)

#### variables.var - Name the suite and add PVs for the program
```iecst
(********************************************************************
 * COPYRIGHT --  MyAutomation-IT
 ********************************************************************
 * Program: Tests_Shooter_C
 * File: variables.var
 * Author: Raivo Berends
 ********************************************************************
 * Local variables of program Tests_Shooter_C
 ********************************************************************)
(*Describe the test*)
VAR
	Testsuite : UtMgrTestSuite := (Name:='Shooter_Tests',Type:=utMgrTEST_TYPE_C);
END_VAR
(*Variables used in the tests*)
VAR
	ShooterFB : FB_Shooter;
	ShooterStruct : UDT_Shooter;
END_VAR
```

#### testSuite.c
```c
/********************************************************************
 * COPYRIGHT - MyAutomation-IT
 ********************************************************************
 * Program: Tests_PaddleMotor_C::testSuite.c
 * Author: Raivo Berends
 * Created: 10-4-2026
 ********************************************************************
 * Test registration and handshake
 ********************************************************************/

#include <bur/plctypes.h>

#ifdef _DEFAULT_INCLUDES
#include <AsDefault.h>
#endif

#include "UnitTest.h"
#include "Library.h"

void _INIT initTestSuite(void)
{
	utInit(&Testsuite);
}

void _CYCLIC cyclicWithTest(void)
{
	utCyclic(&Testsuite);
}

void _EXIT exitTestSuite(void)
{
	utExit(&Testsuite);
}
```

#### autoGeneratedFile.c - Auto generated code - list of all test sets in the program
```c
/*
B+R UnitTest: This is generated code.
Do not edit! Do not move!
Description: UnitTest Testprogramm infrastructure (List of TestSets).
LastUpdated: 2026-05-07 09:31:14Z
By B+R UnitTest Helper Version: 2.0.2.35
*/
#include "UnitTest.h"

UNITTEST_TESTSET_DECLARATION  testSet_Shooter_Disabled;
UNITTEST_TESTSET_DECLARATION  testSet_Shooter_Idle;
UNITTEST_TESTSET_DECLARATION  testSet_Shooter_Shooting;

UNITTEST_TESTSET_FIXTURES(utTestSets)
{
	new_TestSet(testSet_Shooter_Disabled),
	new_TestSet(testSet_Shooter_Idle),
	new_TestSet(testSet_Shooter_Shooting),
};
UNTITTEST_TESTSET_HANDLER();
```

#### testSet_Shooter_Disabled.c
```c
/********************************************************************
 * COPYRIGHT - MyAutoMation-IT
 ********************************************************************
 * Author: Raivo Berends
 ********************************************************************/

#include <bur/plctypes.h>

#ifdef _DEFAULT_INCLUDES
#include <AsDefault.h>
#endif

#include "UnitTest.h"
#include "Library.h"
#include "CommonTypes.h"
#include <string.h>

_SETUP_TEST(void)
{
	ShooterFB.Shooter = &ShooterStruct;
	memset(	ShooterFB.Shooter, 0, sizeof(*ShooterFB.Shooter));
	ShooterFB.Shooter->STS.StateInt = STATE_DISABLED;

	TEST_DONE;
}

_TEST Test_Disabled_SetsDisabledState(void)
{
	ShooterFB.Shooter->STS.StateInt = STATE_DISABLED;

	FB_Shooter(&ShooterFB);

	TEST_ASSERT_EQUAL_INT(1, ShooterFB.Shooter->STS.Disabled);
	TEST_ASSERT_EQUAL_INT(0, ShooterFB.Shooter->STS.Idle);

	TEST_DONE;
}

_TEST Test_Disabled_ResetsHMICommands(void)
{
	ShooterFB.Shooter->STS.StateInt = STATE_DISABLED;

	ShooterFB.Shooter->HMI.Shoot = 1;
	ShooterFB.Shooter->HMI.EnableFan = 1;

	FB_Shooter(&ShooterFB);

	TEST_ASSERT_EQUAL_INT(0, ShooterFB.Shooter->HMI.Shoot);
	TEST_ASSERT_EQUAL_INT(0, ShooterFB.Shooter->HMI.EnableFan);

	TEST_DONE;
}

_TEST Test_Disabled_ResetsControlCommands(void)
{
	ShooterFB.Shooter->STS.StateInt = STATE_DISABLED;

	ShooterFB.Shooter->CS.Shoot = 1;
	ShooterFB.Shooter->CS.EnableFan = 1;
	ShooterFB.Shooter->CS.Interlock = 1;

	FB_Shooter(&ShooterFB);

	TEST_ASSERT_EQUAL_INT(0, ShooterFB.Shooter->CS.Shoot);
	TEST_ASSERT_EQUAL_INT(0, ShooterFB.Shooter->CS.EnableFan);
	TEST_ASSERT_EQUAL_INT(0, ShooterFB.Shooter->CS.Interlock);

	TEST_DONE;
}

_TEST Test_Disabled_ResetsIOOutputs(void)
{
	ShooterFB.Shooter->STS.StateInt = STATE_DISABLED;

	ShooterFB.Shooter->IO.Shoot = 1;
	ShooterFB.Shooter->IO.EnableFan = 1;

	FB_Shooter(&ShooterFB);

	TEST_ASSERT_EQUAL_INT(0, ShooterFB.Shooter->IO.Shoot);
	TEST_ASSERT_EQUAL_INT(0, ShooterFB.Shooter->IO.EnableFan);

	TEST_DONE;
}

_TEST Test_Disabled_ResetsPhysicalOutputs(void)
{
	ShooterFB.Shooter->STS.StateInt = STATE_DISABLED;

	ShooterFB.Shooter->HMI.Shoot = 1;
	ShooterFB.Shooter->HMI.EnableFan = 1;

	FB_Shooter(&ShooterFB);

	TEST_ASSERT_EQUAL_INT(0, ShooterFB.digitalOutput);

	TEST_DONE;
}

_TEST Test_Disabled_TransitionsToIdle(void)
{
	ShooterFB.Shooter->STS.StateInt = STATE_DISABLED;

	ShooterFB.Shooter->CS.Start = 1;
	ShooterFB.Shooter->STS.AlarmActive = 0;
	ShooterFB.Shooter->STS.Interlocked = 0;

	FB_Shooter(&ShooterFB);

	TEST_ASSERT_EQUAL_INT(STATE_IDLE, ShooterFB.Shooter->STS.StateInt);

	TEST_DONE;
}

_TEST Test_Disabled_DoesNotTransitionWhenAlarmActive(void)
{
	ShooterFB.Shooter->STS.StateInt = STATE_DISABLED;

	ShooterFB.Shooter->CS.Start = 1;
	ShooterFB.Shooter->STS.AlarmActive = 1;
	ShooterFB.Shooter->STS.Interlocked = 0;

	FB_Shooter(&ShooterFB);

	TEST_ASSERT_EQUAL_INT(STATE_DISABLED, ShooterFB.Shooter->STS.StateInt);

	TEST_DONE;
}

_TEST Test_Disabled_DoesNotTransitionWhenInterlocked(void)
{
	ShooterFB.Shooter->STS.StateInt = STATE_DISABLED;

	ShooterFB.Shooter->CS.Start = 1;
	ShooterFB.Shooter->STS.AlarmActive = 0;
	ShooterFB.Shooter->STS.Interlocked = 1;

	FB_Shooter(&ShooterFB);

	TEST_ASSERT_EQUAL_INT(STATE_DISABLED, ShooterFB.Shooter->STS.StateInt);

	TEST_DONE;
}

_TEST Test_Disabled_AlarmColourGreen(void)
{
	ShooterFB.Shooter->STS.StateInt = STATE_DISABLED;
	ShooterFB.Shooter->STS.Interlocked = 0;

	FB_Shooter(&ShooterFB);

	TEST_ASSERT_EQUAL_INT(GREEN_COLOUR, ShooterFB.Shooter->STS.AlarmActiveColour);

	TEST_DONE;
}

_TEST Test_Disabled_AlarmColourRed(void)
{
	ShooterFB.Shooter->STS.StateInt = STATE_DISABLED;
	ShooterFB.Shooter->STS.Interlocked = 1;

	FB_Shooter(&ShooterFB);

	TEST_ASSERT_EQUAL_INT(RED_COLOUR, ShooterFB.Shooter->STS.AlarmActiveColour);

	TEST_DONE;
}

_TEST Test_Disabled_StopGameForcesDisabled(void)
{
	ShooterFB.Shooter->STS.StateInt = STATE_IDLE;

	ShooterFB.Shooter->CS.StopGame = 1;
	ShooterFB.Shooter->STS.Interlocked = 0;

	FB_Shooter(&ShooterFB);

	TEST_ASSERT_EQUAL_INT(STATE_DISABLED, ShooterFB.Shooter->STS.StateInt);

	TEST_DONE;
}

_TEST Test_Disabled_StopGameBlockedByInterlock(void)
{
	ShooterFB.Shooter->STS.StateInt = STATE_IDLE;

	ShooterFB.Shooter->CS.StopGame = 1;
	ShooterFB.Shooter->STS.Interlocked = 1;

	FB_Shooter(&ShooterFB);

	TEST_ASSERT_EQUAL_INT(STATE_IDLE, ShooterFB.Shooter->STS.StateInt);

	TEST_DONE;
}

_TEST Test_Disabled_MapsAutoModeToAutoActive(void)
{
	ShooterFB.Shooter->STS.StateInt = STATE_DISABLED;

	ShooterFB.Shooter->CS.AutoMode = 1;

	FB_Shooter(&ShooterFB);

	TEST_ASSERT_EQUAL_INT(1, ShooterFB.Shooter->STS.AutoActive);

	TEST_DONE;
}

/*
B+R UnitTest: This is generated code.
Do not edit! Do not move!
Description: UnitTest Testprogramm infrastructure (TestSet).
LastUpdated: 2026-05-07 09:17:24Z
By B+R UnitTest Helper Version: 2.0.2.35
*/
UNITTEST_FIXTURES(fixtures)
{
	new_TestFixture("Test_Disabled_SetsDisabledState", Test_Disabled_SetsDisabledState),
	new_TestFixture("Test_Disabled_ResetsHMICommands", Test_Disabled_ResetsHMICommands),
	new_TestFixture("Test_Disabled_ResetsControlCommands", Test_Disabled_ResetsControlCommands),
	new_TestFixture("Test_Disabled_ResetsIOOutputs", Test_Disabled_ResetsIOOutputs),
	new_TestFixture("Test_Disabled_ResetsPhysicalOutputs", Test_Disabled_ResetsPhysicalOutputs),
	new_TestFixture("Test_Disabled_TransitionsToIdle", Test_Disabled_TransitionsToIdle),
	new_TestFixture("Test_Disabled_DoesNotTransitionWhenAlarmActive", Test_Disabled_DoesNotTransitionWhenAlarmActive),
	new_TestFixture("Test_Disabled_DoesNotTransitionWhenInterlocked", Test_Disabled_DoesNotTransitionWhenInterlocked),
	new_TestFixture("Test_Disabled_AlarmColourGreen", Test_Disabled_AlarmColourGreen),
	new_TestFixture("Test_Disabled_AlarmColourRed", Test_Disabled_AlarmColourRed),
	new_TestFixture("Test_Disabled_StopGameForcesDisabled", Test_Disabled_StopGameForcesDisabled),
	new_TestFixture("Test_Disabled_StopGameBlockedByInterlock", Test_Disabled_StopGameBlockedByInterlock),
	new_TestFixture("Test_Disabled_MapsAutoModeToAutoActive", Test_Disabled_MapsAutoModeToAutoActive),
};

UNITTEST_CALLER_COMPLETE_EXPLICIT(testSet_Shooter_Disabled, "testSet_Shooter_Disabled", setupTest, 0, fixtures, 0, 0, 0);
```

#### testSet_Shooter_Idle.c
```c
/********************************************************************
 * COPYRIGHT - MyAutoMation-IT
 ********************************************************************
 * Author: Raivo Berends
 ********************************************************************/

#include <bur/plctypes.h>

#ifdef _DEFAULT_INCLUDES
#include <AsDefault.h>
#endif

#include "UnitTest.h"
#include "Library.h"
#include "CommonTypes.h"
#include <string.h>

_SETUP_TEST(void)
{
	ShooterFB.Shooter = &ShooterStruct;
	memset(	ShooterFB.Shooter, 0, sizeof(*ShooterFB.Shooter));
	ShooterFB.Shooter->STS.StateInt = STATE_IDLE;

	TEST_DONE;
}

_TEST Test_Idle_SetsIdleState(void)
{
	ShooterFB.Shooter->STS.StateInt = STATE_IDLE;

	FB_Shooter(&ShooterFB);

	TEST_ASSERT_EQUAL_INT(1, ShooterFB.Shooter->STS.Idle);
	TEST_ASSERT_EQUAL_INT(0, ShooterFB.Shooter->STS.Disabled);
	TEST_ASSERT_EQUAL_INT(0, ShooterFB.Shooter->STS.Shooting);

	TEST_DONE;
}

_TEST Test_Idle_ResetsInterlockCommand(void)
{
	ShooterFB.Shooter->STS.StateInt = STATE_IDLE;

	ShooterFB.Shooter->CS.Interlock = 1;
	ShooterFB.Shooter->HMI.EnableFan = 1;

	FB_Shooter(&ShooterFB);

	TEST_ASSERT_EQUAL_INT(0, ShooterFB.Shooter->CS.Interlock);

	TEST_DONE;
}

_TEST Test_Idle_AutoModeResetsHMIShoot(void)
{
	ShooterFB.Shooter->STS.StateInt = STATE_IDLE;

	ShooterFB.Shooter->STS.AutoActive = 1;
	ShooterFB.Shooter->HMI.Shoot = 1;

	FB_Shooter(&ShooterFB);

	TEST_ASSERT_EQUAL_INT(0, ShooterFB.Shooter->HMI.Shoot);

	TEST_DONE;
}

_TEST Test_Idle_InterlockSetWhenFanDisabled(void)
{
	ShooterFB.Shooter->STS.StateInt = STATE_IDLE;

	ShooterFB.Shooter->STS.AutoActive = 0;
	ShooterFB.Shooter->HMI.EnableFan = 0;

	FB_Shooter(&ShooterFB);

	TEST_ASSERT_EQUAL_INT(1, ShooterFB.Shooter->CS.Interlock);

	TEST_DONE;
}

_TEST Test_Idle_NoInterlockWhenFanEnabled(void)
{
	ShooterFB.Shooter->STS.StateInt = STATE_IDLE;

	ShooterFB.Shooter->STS.AutoActive = 0;
	ShooterFB.Shooter->HMI.EnableFan = 1;

	FB_Shooter(&ShooterFB);

	TEST_ASSERT_EQUAL_INT(0, ShooterFB.Shooter->CS.Interlock);

	TEST_DONE;
}

_TEST Test_Idle_ResetsShootCommand(void)
{
	ShooterFB.Shooter->STS.StateInt = STATE_IDLE;

	ShooterFB.Shooter->STS.AutoActive = 0;
	ShooterFB.Shooter->CS.Shoot = 1;

	FB_Shooter(&ShooterFB);

	TEST_ASSERT_EQUAL_INT(0, ShooterFB.Shooter->CS.Shoot);

	TEST_DONE;
}

_TEST Test_Idle_TransitionsToShootingFromHMI(void)
{
	ShooterFB.Shooter->STS.StateInt = STATE_IDLE;

	ShooterFB.Shooter->HMI.Shoot = 1;
	ShooterFB.Shooter->CS.Shoot = 0;

	ShooterFB.Shooter->STS.AlarmActive = 0;
	ShooterFB.Shooter->STS.Interlocked = 0;

	FB_Shooter(&ShooterFB);

	TEST_ASSERT_EQUAL_INT(STATE_SHOOTING, ShooterFB.Shooter->STS.StateInt);

	TEST_DONE;
}

_TEST Test_Idle_TransitionsToShootingFromControl(void)
{
	ShooterFB.Shooter->STS.StateInt = STATE_IDLE;

	ShooterFB.Shooter->HMI.Shoot = 0;
	ShooterFB.Shooter->CS.Shoot = 1;

	ShooterFB.Shooter->STS.AlarmActive = 0;
	ShooterFB.Shooter->STS.Interlocked = 0;
	ShooterFB.Shooter->STS.AutoActive = 1;

	FB_Shooter(&ShooterFB);

	TEST_ASSERT_EQUAL_INT(STATE_SHOOTING, ShooterFB.Shooter->STS.StateInt);

	TEST_DONE;
}

_TEST Test_Idle_DoesNotTransitionWhenAlarmActive(void)
{
	ShooterFB.Shooter->STS.StateInt = STATE_IDLE;

	ShooterFB.Shooter->HMI.Shoot = 1;
	ShooterFB.Shooter->CS.Shoot = 0;

	ShooterFB.Shooter->STS.AlarmActive = 1;
	ShooterFB.Shooter->STS.Interlocked = 0;

	FB_Shooter(&ShooterFB);

	TEST_ASSERT_EQUAL_INT(STATE_IDLE, ShooterFB.Shooter->STS.StateInt);

	TEST_DONE;
}

_TEST Test_Idle_DoesNotTransitionWhenInterlocked(void)
{
	ShooterFB.Shooter->STS.StateInt = STATE_IDLE;

	ShooterFB.Shooter->HMI.Shoot = 1;
	ShooterFB.Shooter->CS.Shoot = 0;

	ShooterFB.Shooter->STS.AlarmActive = 0;
	ShooterFB.Shooter->STS.Interlocked = 1;

	FB_Shooter(&ShooterFB);

	TEST_ASSERT_EQUAL_INT(STATE_IDLE, ShooterFB.Shooter->STS.StateInt);

	TEST_DONE;
}

_TEST Test_Idle_SetsShootOutput(void)
{
	ShooterFB.Shooter->STS.StateInt = STATE_IDLE;

	ShooterFB.Shooter->HMI.Shoot = 1;
	ShooterFB.Shooter->CS.Shoot = 0;

	ShooterFB.Shooter->STS.AlarmActive = 0;
	ShooterFB.Shooter->STS.Interlocked = 0;

	FB_Shooter(&ShooterFB);

	TEST_ASSERT_EQUAL_INT(1, ShooterFB.Shooter->IO.Shoot);

	TEST_DONE;
}

_TEST Test_Idle_BlocksShootOutputWhenInterlocked(void)
{
	ShooterFB.Shooter->STS.StateInt = STATE_IDLE;

	ShooterFB.Shooter->HMI.Shoot = 1;
	ShooterFB.Shooter->CS.Shoot = 0;

	ShooterFB.Shooter->STS.Interlocked = 1;

	FB_Shooter(&ShooterFB);

	TEST_ASSERT_EQUAL_INT(0, ShooterFB.Shooter->IO.Shoot);

	TEST_DONE;
}

_TEST Test_Idle_BlocksShootOutputWhenAlarmActive(void)
{
	ShooterFB.Shooter->STS.StateInt = STATE_IDLE;

	ShooterFB.Shooter->HMI.Shoot = 1;
	ShooterFB.Shooter->CS.Shoot = 0;

	ShooterFB.Shooter->STS.AlarmActive = 1;

	FB_Shooter(&ShooterFB);

	TEST_ASSERT_EQUAL_INT(0, ShooterFB.Shooter->IO.Shoot);

	TEST_DONE;
}

_TEST Test_Idle_EnableFanOutputMapping(void)
{
	ShooterFB.Shooter->STS.StateInt = STATE_IDLE;

	ShooterFB.Shooter->HMI.EnableFan = 1;
	ShooterFB.Shooter->CS.EnableFan = 0;

	FB_Shooter(&ShooterFB);

	TEST_ASSERT_EQUAL_INT(1, ShooterFB.Shooter->IO.EnableFan);

	TEST_DONE;
}

_TEST Test_Idle_DigitalOutputMapping(void)
{
	ShooterFB.Shooter->STS.StateInt = STATE_IDLE;

	ShooterFB.Shooter->HMI.Shoot = 1;
	ShooterFB.Shooter->HMI.EnableFan = 1;

	ShooterFB.Shooter->STS.AlarmActive = 0;
	ShooterFB.Shooter->STS.Interlocked = 0;

	FB_Shooter(&ShooterFB);

	TEST_ASSERT_EQUAL_INT((1 << SHOOT_OUTPUT_BIT) | (1 << FAN_OUTPUT_BIT), ShooterFB.digitalOutput);

	TEST_DONE;
}

_TEST Test_Idle_MapsInterlockStatus(void)
{
	ShooterFB.Shooter->STS.StateInt = STATE_IDLE;

	ShooterFB.Shooter->CS.Interlock = 1;

	FB_Shooter(&ShooterFB);

	TEST_ASSERT_EQUAL_INT(1, ShooterFB.Shooter->STS.Interlocked);

	TEST_DONE;
}

_TEST Test_Idle_MapsAutoModeToAutoActive(void)
{
	ShooterFB.Shooter->STS.StateInt = STATE_IDLE;

	ShooterFB.Shooter->CS.AutoMode = 1;

	FB_Shooter(&ShooterFB);

	TEST_ASSERT_EQUAL_INT(1, ShooterFB.Shooter->STS.AutoActive);

	TEST_DONE;
}

/*
B+R UnitTest: This is generated code.
Do not edit! Do not move!
Description: UnitTest Testprogramm infrastructure (TestSet).
LastUpdated: 2026-05-07 09:25:21Z
By B+R UnitTest Helper Version: 2.0.2.35
*/
UNITTEST_FIXTURES(fixtures)
{
	new_TestFixture("Test_Idle_SetsIdleState", Test_Idle_SetsIdleState),
	new_TestFixture("Test_Idle_ResetsInterlockCommand", Test_Idle_ResetsInterlockCommand),
	new_TestFixture("Test_Idle_AutoModeResetsHMIShoot", Test_Idle_AutoModeResetsHMIShoot),
	new_TestFixture("Test_Idle_InterlockSetWhenFanDisabled", Test_Idle_InterlockSetWhenFanDisabled),
	new_TestFixture("Test_Idle_NoInterlockWhenFanEnabled", Test_Idle_NoInterlockWhenFanEnabled),
	new_TestFixture("Test_Idle_ResetsShootCommand", Test_Idle_ResetsShootCommand),
	new_TestFixture("Test_Idle_TransitionsToShootingFromHMI", Test_Idle_TransitionsToShootingFromHMI),
	new_TestFixture("Test_Idle_TransitionsToShootingFromControl", Test_Idle_TransitionsToShootingFromControl),
	new_TestFixture("Test_Idle_DoesNotTransitionWhenAlarmActive", Test_Idle_DoesNotTransitionWhenAlarmActive),
	new_TestFixture("Test_Idle_DoesNotTransitionWhenInterlocked", Test_Idle_DoesNotTransitionWhenInterlocked),
	new_TestFixture("Test_Idle_SetsShootOutput", Test_Idle_SetsShootOutput),
	new_TestFixture("Test_Idle_BlocksShootOutputWhenInterlocked", Test_Idle_BlocksShootOutputWhenInterlocked),
	new_TestFixture("Test_Idle_BlocksShootOutputWhenAlarmActive", Test_Idle_BlocksShootOutputWhenAlarmActive),
	new_TestFixture("Test_Idle_EnableFanOutputMapping", Test_Idle_EnableFanOutputMapping),
	new_TestFixture("Test_Idle_DigitalOutputMapping", Test_Idle_DigitalOutputMapping),
	new_TestFixture("Test_Idle_MapsInterlockStatus", Test_Idle_MapsInterlockStatus),
	new_TestFixture("Test_Idle_MapsAutoModeToAutoActive", Test_Idle_MapsAutoModeToAutoActive),
};

UNITTEST_CALLER_COMPLETE_EXPLICIT(testSet_Shooter_Idle, "testSet_Shooter_Idle", setupTest, 0, fixtures, 0, 0, 0);
```

#### testSet_Shooter_Shooting.c
```c
/********************************************************************
 * COPYRIGHT - MyAutoMation-IT
 ********************************************************************
 * Author: Raivo Berends
 ********************************************************************/

#include <bur/plctypes.h>

#ifdef _DEFAULT_INCLUDES
#include <AsDefault.h>
#endif

#include "UnitTest.h"
#include "Library.h"
#include "CommonTypes.h"
#include <string.h>

_SETUP_TEST(void)
{
	ShooterFB.Shooter = &ShooterStruct;
	memset(	ShooterFB.Shooter, 0, sizeof(*ShooterFB.Shooter));
	ShooterFB.Shooter->STS.StateInt = STATE_SHOOTING;

	TEST_DONE;
}

_TEST Test_Shooting_SetsShootingState(void)
{
	ShooterFB.Shooter->STS.StateInt = STATE_SHOOTING;

	FB_Shooter(&ShooterFB);

	TEST_ASSERT_EQUAL_INT(1, ShooterFB.Shooter->STS.Shooting);

	TEST_DONE;
}

_TEST Test_Shooting_ReturnsToIdleWhenNoRequest(void)
{
	ShooterFB.Shooter->STS.StateInt = STATE_SHOOTING;

	ShooterFB.Shooter->CS.Shoot = 0;
	ShooterFB.Shooter->HMI.Shoot = 0;

	ShooterFB.Shooter->STS.AlarmActive = 0;
	ShooterFB.Shooter->STS.Interlocked = 0;

	FB_Shooter(&ShooterFB);

	TEST_ASSERT_EQUAL_INT(STATE_IDLE, ShooterFB.Shooter->STS.StateInt);

	TEST_DONE;
}

_TEST Test_Shooting_DoesNotReturnToIdleWhenHMIRequestExists(void)
{
	ShooterFB.Shooter->STS.StateInt = STATE_SHOOTING;

	ShooterFB.Shooter->CS.Shoot = 0;
	ShooterFB.Shooter->HMI.Shoot = 1;

	FB_Shooter(&ShooterFB);

	TEST_ASSERT_EQUAL_INT(STATE_SHOOTING, ShooterFB.Shooter->STS.StateInt);

	TEST_DONE;
}

_TEST Test_Shooting_DoesNotReturnToIdleWhenCSRequestExists(void)
{
	ShooterFB.Shooter->STS.StateInt = STATE_SHOOTING;

	ShooterFB.Shooter->CS.Shoot = 1;
	ShooterFB.Shooter->HMI.Shoot = 0;

	FB_Shooter(&ShooterFB);

	TEST_ASSERT_EQUAL_INT(STATE_SHOOTING, ShooterFB.Shooter->STS.StateInt);

	TEST_DONE;
}

_TEST Test_Shooting_DoesNotReturnToIdleWhenAlarmActive(void)
{
	ShooterFB.Shooter->STS.StateInt = STATE_SHOOTING;

	ShooterFB.Shooter->CS.Shoot = 0;
	ShooterFB.Shooter->HMI.Shoot = 0;

	ShooterFB.Shooter->STS.AlarmActive = 1;

	FB_Shooter(&ShooterFB);

	TEST_ASSERT_EQUAL_INT(STATE_SHOOTING, ShooterFB.Shooter->STS.StateInt);

	TEST_DONE;
}

_TEST Test_Shooting_DoesNotReturnToIdleWhenInterlocked(void)
{
	ShooterFB.Shooter->STS.StateInt = STATE_SHOOTING;

	ShooterFB.Shooter->CS.Shoot = 0;
	ShooterFB.Shooter->HMI.Shoot = 0;

	ShooterFB.Shooter->STS.Interlocked = 1;

	FB_Shooter(&ShooterFB);

	TEST_ASSERT_EQUAL_INT(STATE_SHOOTING, ShooterFB.Shooter->STS.StateInt);

	TEST_DONE;
}

_TEST Test_Shooting_OutputNotUpdatedWhenUnsafe(void)
{
	ShooterFB.Shooter->STS.StateInt = STATE_SHOOTING;

	ShooterFB.Shooter->STS.Interlocked = 1;

	ShooterFB.Shooter->HMI.Shoot = 1;
	ShooterFB.Shooter->CS.Shoot = 0;

	FB_Shooter(&ShooterFB);

	TEST_ASSERT_EQUAL_INT(0, ShooterFB.Shooter->IO.Shoot);

	TEST_DONE;
}

_TEST Test_Shooting_OutputMappingActiveWhenSafe(void)
{
	ShooterFB.Shooter->STS.StateInt = STATE_SHOOTING;

	ShooterFB.Shooter->STS.Interlocked = 0;
	ShooterFB.Shooter->STS.AlarmActive = 0;

	ShooterFB.Shooter->HMI.Shoot = 1;
	ShooterFB.Shooter->CS.Shoot = 0;

	FB_Shooter(&ShooterFB);

	TEST_ASSERT_EQUAL_INT(1, ShooterFB.Shooter->IO.Shoot);

	TEST_DONE;
}

/*
B+R UnitTest: This is generated code.
Do not edit! Do not move!
Description: UnitTest Testprogramm infrastructure (TestSet).
LastUpdated: 2026-05-07 09:31:14Z
By B+R UnitTest Helper Version: 2.0.2.35
*/
UNITTEST_FIXTURES(fixtures)
{
	new_TestFixture("Test_Shooting_SetsShootingState", Test_Shooting_SetsShootingState),
	new_TestFixture("Test_Shooting_ReturnsToIdleWhenNoRequest", Test_Shooting_ReturnsToIdleWhenNoRequest),
	new_TestFixture("Test_Shooting_DoesNotReturnToIdleWhenHMIRequestExists", Test_Shooting_DoesNotReturnToIdleWhenHMIRequestExists),
	new_TestFixture("Test_Shooting_DoesNotReturnToIdleWhenCSRequestExists", Test_Shooting_DoesNotReturnToIdleWhenCSRequestExists),
	new_TestFixture("Test_Shooting_DoesNotReturnToIdleWhenAlarmActive", Test_Shooting_DoesNotReturnToIdleWhenAlarmActive),
	new_TestFixture("Test_Shooting_DoesNotReturnToIdleWhenInterlocked", Test_Shooting_DoesNotReturnToIdleWhenInterlocked),
	new_TestFixture("Test_Shooting_OutputNotUpdatedWhenUnsafe", Test_Shooting_OutputNotUpdatedWhenUnsafe),
	new_TestFixture("Test_Shooting_OutputMappingActiveWhenSafe", Test_Shooting_OutputMappingActiveWhenSafe),
};

UNITTEST_CALLER_COMPLETE_EXPLICIT(testSet_Shooter_Shooting, "testSet_Shooter_Shooting", setupTest, 0, fixtures, 0, 0, 0);
```

### Program Logical/UnitTests/HelperTool_Supported/Tests_PaddleMotor_C (ANSIC)

#### variables.var - Name the suite and add PVs for the program
```iecst
(********************************************************************
 * COPYRIGHT --  MyAutomation-IT
 ********************************************************************
 * Program: Tests_PaddleMotor_C
 * File: variables.var
 * Author: Raivo Berends
 ********************************************************************
 * Local variables of program Tests_PaddleMotor_C
 ********************************************************************)
(*Describe the test*)
VAR
	Testsuite : UtMgrTestSuite := (Name:='PaddleMotor_Tests',Type:=utMgrTEST_TYPE_C);
END_VAR
(*Variables used in the tests*)
VAR
	PaddleMotorFB : FB_PaddleMotor;
	PaddleMotorStruct : UDT_PaddleMotor;
END_VAR
```

#### autoGeneratedFile.c - Auto generated code - list of all test sets in the program
```c
/*
B+R UnitTest: This is generated code.
Do not edit! Do not move!
Description: UnitTest Testprogramm infrastructure (List of TestSets).
LastUpdated: 2026-04-14 09:06:48Z
By B+R UnitTest Helper Version: 2.0.2.35
*/
#include "UnitTest.h"

UNITTEST_TESTSET_DECLARATION  testSet_PaddleMotor_Disabled;
UNITTEST_TESTSET_DECLARATION  testSet_PaddleMotor_Initializing;

UNITTEST_TESTSET_FIXTURES(utTestSets)
{
	new_TestSet(testSet_PaddleMotor_Disabled),
	new_TestSet(testSet_PaddleMotor_Initializing),
};
UNTITTEST_TESTSET_HANDLER();
```

#### testSet_PaddleMotor_Disabled.c
```c
/********************************************************************
 * COPYRIGHT --
 ********************************************************************
 * Program: -
 * Author:
 * Created:
 ********************************************************************
 * Tests for ...
 ********************************************************************/

#include <bur/plctypes.h>

#ifdef _DEFAULT_INCLUDES
#include <AsDefault.h>
#endif

#include "UnitTest.h"
#include "Library.h"

#define STATE_DISABLED 0
#define STATE_INITIALIZING 10

_TEST test_Disabled_State_DefaultBehavior(void)
{
	PaddleMotorFB.digitalInput = 0;
	PaddleMotorFB.PaddleMotor = &PaddleMotorStruct;

	// Set beginstate
	PaddleMotorFB.PaddleMotor->STS.StateInt = STATE_DISABLED;

	// Setting signals that have to be reset
	PaddleMotorFB.PaddleMotor->CS.Power = 1;
	PaddleMotorFB.PaddleMotor->CS.Home = 1;
	PaddleMotorFB.PaddleMotor->CS.MoveJogNeg = 1;
	PaddleMotorFB.PaddleMotor->CS.MoveJogPos = 1;
	PaddleMotorFB.PaddleMotor->CS.MoveAbsolute = 1;

	PaddleMotorFB.PaddleMotor->HMI.MoveJogNeg = 1;
	PaddleMotorFB.PaddleMotor->HMI.MoveJogPos = 1;

	PaddleMotorFB.PaddleMotor->STS.TimerStarted = 1;
	PaddleMotorFB.PaddleMotor->STS.TimerEnded = 1;
	PaddleMotorFB.PaddleMotor->STS.ReferencePosition = 1234;
	PaddleMotorFB.PaddleMotor->STS.ReferenceSet = 1;

	FB_PaddleMotor(&PaddleMotorFB);

	TEST_ASSERT_EQUAL_INT(1, PaddleMotorFB.PaddleMotor->STS.Disabled);

	TEST_ASSERT_EQUAL_INT(0, PaddleMotorFB.PaddleMotor->CS.Power);
	TEST_ASSERT_EQUAL_INT(0, PaddleMotorFB.PaddleMotor->CS.Home);
	TEST_ASSERT_EQUAL_INT(0, PaddleMotorFB.PaddleMotor->CS.MoveJogNeg);
	TEST_ASSERT_EQUAL_INT(0, PaddleMotorFB.PaddleMotor->CS.MoveJogPos);
	TEST_ASSERT_EQUAL_INT(0, PaddleMotorFB.PaddleMotor->CS.MoveAbsolute);

	TEST_ASSERT_EQUAL_INT(0, PaddleMotorFB.PaddleMotor->HMI.MoveJogNeg);
	TEST_ASSERT_EQUAL_INT(0, PaddleMotorFB.PaddleMotor->HMI.MoveJogPos);

	TEST_ASSERT_EQUAL_INT(0, PaddleMotorFB.PaddleMotor->STS.TimerStarted);
	TEST_ASSERT_EQUAL_INT(0, PaddleMotorFB.PaddleMotor->STS.TimerEnded);
	TEST_ASSERT_EQUAL_INT(0, PaddleMotorFB.PaddleMotor->STS.ReferencePosition);
	TEST_ASSERT_EQUAL_INT(0, PaddleMotorFB.PaddleMotor->STS.ReferenceSet);

	TEST_DONE;
}

_TEST test_Disabled_NoInitialize_StaysDisabled(void)
{
	PaddleMotorFB.PaddleMotor = &PaddleMotorStruct;

	PaddleMotorFB.PaddleMotor->STS.StateInt = STATE_DISABLED;
	PaddleMotorFB.PaddleMotor->CS.Initialize = 0;
	PaddleMotorFB.PaddleMotor->STS.AlarmActive = 0;
	PaddleMotorFB.PaddleMotor->STS.Interlocked = 0;

	FB_PaddleMotor(&PaddleMotorFB);

	TEST_ASSERT_EQUAL_INT(STATE_DISABLED, PaddleMotorFB.PaddleMotor->STS.StateInt);

	TEST_DONE;
}

_TEST test_Disabled_ToInitializing(void)
{
	PaddleMotorFB.PaddleMotor = &PaddleMotorStruct;

	PaddleMotorFB.PaddleMotor->STS.StateInt = STATE_DISABLED;
	PaddleMotorFB.PaddleMotor->CS.Initialize = 1;
	PaddleMotorFB.PaddleMotor->STS.AlarmActive = 0;
	PaddleMotorFB.PaddleMotor->STS.Interlocked = 0;

	FB_PaddleMotor(&PaddleMotorFB);

	TEST_ASSERT_EQUAL_INT(STATE_INITIALIZING, PaddleMotorFB.PaddleMotor->STS.StateInt);

	TEST_DONE;
}

_TEST test_Disabled_NoTransition_WhenAlarm(void)
{
	PaddleMotorFB.PaddleMotor = &PaddleMotorStruct;

	PaddleMotorFB.PaddleMotor->STS.StateInt = STATE_DISABLED;
	PaddleMotorFB.PaddleMotor->CS.Initialize = 1;
	PaddleMotorFB.PaddleMotor->STS.AlarmActive = 1;
	PaddleMotorFB.PaddleMotor->STS.Interlocked = 0;

	FB_PaddleMotor(&PaddleMotorFB);

	TEST_ASSERT_EQUAL_INT(STATE_DISABLED, PaddleMotorFB.PaddleMotor->STS.StateInt);

	TEST_DONE;
}

_TEST test_Disabled_NoTransition_WhenInterlocked(void)
{
	PaddleMotorFB.PaddleMotor = &PaddleMotorStruct;

	PaddleMotorFB.PaddleMotor->STS.StateInt = STATE_DISABLED;
	PaddleMotorFB.PaddleMotor->CS.Initialize = 1;
	PaddleMotorFB.PaddleMotor->STS.AlarmActive = 0;
	PaddleMotorFB.PaddleMotor->STS.Interlocked = 1;

	FB_PaddleMotor(&PaddleMotorFB);

	TEST_ASSERT_EQUAL_INT(STATE_DISABLED, PaddleMotorFB.PaddleMotor->STS.StateInt);

	TEST_DONE;
}

/*
B+R UnitTest: This is generated code.
Do not edit! Do not move!
Description: UnitTest Testprogramm infrastructure (TestSet).
LastUpdated: 2026-04-14 09:02:57Z
By B+R UnitTest Helper Version: 2.0.2.35
*/
UNITTEST_FIXTURES(fixtures)
{
	new_TestFixture("test_Disabled_State_DefaultBehavior", test_Disabled_State_DefaultBehavior),
	new_TestFixture("test_Disabled_NoInitialize_StaysDisabled", test_Disabled_NoInitialize_StaysDisabled),
	new_TestFixture("test_Disabled_ToInitializing", test_Disabled_ToInitializing),
	new_TestFixture("test_Disabled_NoTransition_WhenAlarm", test_Disabled_NoTransition_WhenAlarm),
	new_TestFixture("test_Disabled_NoTransition_WhenInterlocked", test_Disabled_NoTransition_WhenInterlocked),
};

UNITTEST_CALLER_COMPLETE_EXPLICIT(testSet_PaddleMotor_Disabled, "testSet_PaddleMotor_Disabled", 0, 0, fixtures, 0, 0, 0);
```

#### testSet_PaddleMotor_Initializing.c
```c
/********************************************************************
 * COPYRIGHT --
 ********************************************************************
 * Program: -
 * Author:
 * Created:
 ********************************************************************
 * Tests for ...
 ********************************************************************/

#include <bur/plctypes.h>

#ifdef _DEFAULT_INCLUDES
#include <AsDefault.h>
#endif

#include "UnitTest.h"
#include "Library.h"

#define STATE_DISABLED 0
#define STATE_INITIALIZING 10
#define STATE_IDLE 20

#define MAX_ACC_DEC 40000
#define MIDDLE_POSITION 1450
#define ENDBUTTON_BITMASK 0x2

_TEST test_Initializing_SetsParameters(void)
{
	PaddleMotorFB.PaddleMotor = &PaddleMotorStruct;

	PaddleMotorFB.PaddleMotor->STS.StateInt = STATE_INITIALIZING;

	FB_PaddleMotor(&PaddleMotorFB);

	TEST_ASSERT_EQUAL_INT(1, PaddleMotorFB.PaddleMotor->STS.Initializing);
	TEST_ASSERT_EQUAL_INT(0, PaddleMotorFB.PaddleMotor->STS.Disabled);

	TEST_ASSERT_EQUAL_INT(MAX_ACC_DEC, PaddleMotorFB.PaddleMotor->PAR.Acceleration);
	TEST_ASSERT_EQUAL_INT(MAX_ACC_DEC, PaddleMotorFB.PaddleMotor->PAR.Deceleration);
	TEST_ASSERT_EQUAL_INT(1000, PaddleMotorFB.PaddleMotor->PAR.JogVelocity);
	TEST_ASSERT_EQUAL_INT(1000, PaddleMotorFB.PaddleMotor->PAR.Velocity);

	TEST_ASSERT_EQUAL_INT(1, PaddleMotorFB.PaddleMotor->CS.Power);
	TEST_ASSERT_EQUAL_INT(0, PaddleMotorFB.PaddleMotor->CS.Stop);

	TEST_DONE;
}

_TEST test_Initializing_StartsHoming(void)
{
	PaddleMotorFB.PaddleMotor = &PaddleMotorStruct;

	PaddleMotorFB.digitalInput = 0; // EndButton = 1
	PaddleMotorFB.PaddleMotor->STS.StateInt = STATE_INITIALIZING;
	PaddleMotorFB.PaddleMotor->STS.EndButtonHit = 0;

	FB_PaddleMotor(&PaddleMotorFB);

	TEST_ASSERT_EQUAL_INT(1, PaddleMotorFB.PaddleMotor->CS.Home);
	TEST_ASSERT_EQUAL_INT(1, PaddleMotorFB.PaddleMotor->STS.TimerStarted);

	TEST_DONE;
}

_TEST test_Initializing_EndButtonHit(void)
{
	PaddleMotorFB.PaddleMotor = &PaddleMotorStruct;

	//Making EndButton active
	PaddleMotorFB.digitalInput = 0x1; //EndButton pressed, 2nd bit = 0

	PaddleMotorFB.PaddleMotor->STS.StateInt = STATE_INITIALIZING;
	PaddleMotorFB.PaddleMotor->STS.EndButtonHit = 0;

	FB_PaddleMotor(&PaddleMotorFB);

	TEST_ASSERT_EQUAL_INT(1, PaddleMotorFB.PaddleMotor->STS.EndButtonHit);
	TEST_ASSERT_EQUAL_INT(1, PaddleMotorFB.PaddleMotor->CS.Home);
	TEST_ASSERT_EQUAL_INT(0, PaddleMotorFB.PaddleMotor->CS.MoveJogPos);

	TEST_DONE;
}

_TEST test_Initializing_ToIdle(void)
{
	PaddleMotorFB.PaddleMotor = &PaddleMotorStruct;

	PaddleMotorFB.PaddleMotor->STS.StateInt = STATE_INITIALIZING;
	PaddleMotorFB.PaddleMotor->STS.EndButtonHit = 1;
	PaddleMotorFB.PaddleMotor->STS.TimerEnded = 1;
	PaddleMotorFB.PaddleMotor->STS.ReferenceSet = 1;

	//PaddleMotorFB.PaddleMotor->STS.ReferencePosition = 3000;
	PaddleMotorFB.PaddleMotor->PAR.Position = 3000;
	PaddleMotorFB.PaddleMotor->STS.ActPosition = 3000;

	PaddleMotorFB.PaddleMotor->STS.AlarmActive = 0;
	PaddleMotorFB.PaddleMotor->STS.Interlocked = 0;

	FB_PaddleMotor(&PaddleMotorFB);

	TEST_ASSERT_EQUAL_INT(STATE_IDLE, PaddleMotorFB.PaddleMotor->STS.StateInt);
	TEST_ASSERT_EQUAL_INT(0, PaddleMotorFB.PaddleMotor->CS.MoveAbsolute);

	TEST_DONE;
}

_TEST test_Initializing_ReferencePosition(void)
{
	PaddleMotorFB.PaddleMotor = &PaddleMotorStruct;

	PaddleMotorFB.PaddleMotor->STS.StateInt = STATE_INITIALIZING;
	PaddleMotorFB.PaddleMotor->STS.EndButtonHit = 1;
	PaddleMotorFB.PaddleMotor->STS.TimerEnded = 1;
	PaddleMotorFB.PaddleMotor->STS.ReferenceSet = 0;

	PaddleMotorFB.PaddleMotor->STS.ActPosition = 5000;

	FB_PaddleMotor(&PaddleMotorFB);

	TEST_ASSERT_EQUAL_INT(5000, PaddleMotorFB.PaddleMotor->STS.ReferencePosition);

	TEST_DONE;
}

_TEST test_Initializing_StartMoveAbsolute(void)
{
	PaddleMotorFB.PaddleMotor = &PaddleMotorStruct;

	PaddleMotorFB.PaddleMotor->STS.StateInt = STATE_INITIALIZING;
	PaddleMotorFB.PaddleMotor->STS.EndButtonHit = 1;
	PaddleMotorFB.PaddleMotor->STS.TimerEnded = 1;
	PaddleMotorFB.PaddleMotor->STS.ReferenceSet = 0;

	PaddleMotorFB.PaddleMotor->STS.ActPosition = 4000;

	FB_PaddleMotor(&PaddleMotorFB);

	TEST_ASSERT_EQUAL_INT(1, PaddleMotorFB.PaddleMotor->CS.MoveAbsolute);

	TEST_DONE;
}

_TEST test_Initializing_TargetPosition(void)
{
	PaddleMotorFB.PaddleMotor = &PaddleMotorStruct;

	PaddleMotorFB.PaddleMotor->STS.StateInt = STATE_INITIALIZING;
	PaddleMotorFB.PaddleMotor->STS.EndButtonHit = 1;
	PaddleMotorFB.PaddleMotor->STS.TimerEnded = 1;
	PaddleMotorFB.PaddleMotor->STS.ReferenceSet = 0;

	PaddleMotorFB.PaddleMotor->STS.ActPosition = 5000;

	FB_PaddleMotor(&PaddleMotorFB);

	TEST_ASSERT_EQUAL_INT(5000 - MIDDLE_POSITION, PaddleMotorFB.PaddleMotor->PAR.Position);

	TEST_DONE;
}

/*
B+R UnitTest: This is generated code.
Do not edit! Do not move!
Description: UnitTest Testprogramm infrastructure (TestSet).
LastUpdated: 2026-04-14 09:36:22Z
By B+R UnitTest Helper Version: 2.0.2.35
*/
UNITTEST_FIXTURES(fixtures)
{
	new_TestFixture("test_Initializing_SetsParameters", test_Initializing_SetsParameters),
	new_TestFixture("test_Initializing_StartsHoming", test_Initializing_StartsHoming),
	new_TestFixture("test_Initializing_EndButtonHit", test_Initializing_EndButtonHit),
	new_TestFixture("test_Initializing_ToIdle", test_Initializing_ToIdle),
	new_TestFixture("test_Initializing_ReferencePosition", test_Initializing_ReferencePosition),
	new_TestFixture("test_Initializing_StartMoveAbsolute", test_Initializing_StartMoveAbsolute),
	new_TestFixture("test_Initializing_TargetPosition", test_Initializing_TargetPosition),
};

UNITTEST_CALLER_COMPLETE_EXPLICIT(testSet_PaddleMotor_Initializing, "testSet_PaddleMotor_Initializing", 0, 0, fixtures, 0, 0, 0);
```

### Program Logical/LibACP10MC_SingleAx_C/Basic (ANSIC) - Basic logical control

#### basic.c - cyclic code
```c
/*******************************************************************
 * COPYRIGHT -- Bernecker + Rainer
 ********************************************************************
 * PROGRAM: Basic
 * File: Basic.c
 * Author: Bernecker + Rainer
 * Created: December 01, 2009
 ********************************************************************
 * Implementation of Program Basic
 ********************************************************************/

#ifdef _DEFAULT_INCLUDES
 #include <AsDefault.h>
#endif
#include <string.h>

/* defines of the state-constants */
#define STATE_WAIT              0
#define STATE_POWER_ON          1
#define STATE_HOME              2

#define STATE_READY             10
#define STATE_HALT              11
#define STATE_STOP              12
#define STATE_JOG_POSITIVE      13
#define STATE_JOG_NEGATIVE      14
#define STATE_MOVE_ABSOLUTE     15
#define STATE_MOVE_ADDITIVE     16
#define STATE_MOVE_VELOCITY     17

#define STATE_ERROR_AXIS        100
#define STATE_ERROR             101
#define STATE_ERROR_RESET       102

_INIT void BasicControl_init(void)
{

/* get axis object */
Axis1Obj = (UDINT)&gAxis01;

AxisStep = STATE_WAIT;  /* start step */

BasicControl.Parameter.Velocity              = 1000;  /*velocity for movement*/
BasicControl.Parameter.Acceleration          = 5000;  /*acceleration for movement*/
BasicControl.Parameter.Deceleration          = 5000;  /*deceleration for movement*/
BasicControl.Parameter.JogVelocity           = 400;   /*velocity for jogging */

}

_CYCLIC void BasicControl_cyclic(void)
{

/***************************************************************
        Control Sequence
***************************************************************/

/* status information is read before the step sequencer to attain a shorter reaction time */
/************************ MC_READSTATUS *************************/
MC_ReadStatus_0.Enable = !MC_ReadStatus_0.Error;
MC_ReadStatus_0.Axis = Axis1Obj;
MC_ReadStatus(&MC_ReadStatus_0);
BasicControl.AxisState.Disabled             = MC_ReadStatus_0.Disabled;
BasicControl.AxisState.StandStill           = MC_ReadStatus_0.StandStill;
BasicControl.AxisState.Stopping             = MC_ReadStatus_0.Stopping;
BasicControl.AxisState.Homing               = MC_ReadStatus_0.Homing;
BasicControl.AxisState.DiscreteMotion       = MC_ReadStatus_0.DiscreteMotion;
BasicControl.AxisState.ContinuousMotion     = MC_ReadStatus_0.ContinuousMotion;
BasicControl.AxisState.SynchronizedMotion   = MC_ReadStatus_0.SynchronizedMotion;
BasicControl.AxisState.ErrorStop            = MC_ReadStatus_0.Errorstop;

/********************MC_BR_READDRIVESTATUS***********************/
MC_BR_ReadDriveStatus_0.Enable = !MC_BR_ReadDriveStatus_0.Error;
MC_BR_ReadDriveStatus_0.Axis = Axis1Obj;
MC_BR_ReadDriveStatus_0.AdrDriveStatus = (UDINT)&(BasicControl.Status.DriveStatus);
MC_BR_ReadDriveStatus(&MC_BR_ReadDriveStatus_0);

/******************** MC_READACTUALPOSITION *********************/
MC_ReadActualPosition_0.Enable = (!MC_ReadActualPosition_0.Error);
MC_ReadActualPosition_0.Axis = Axis1Obj;
MC_ReadActualPosition(&MC_ReadActualPosition_0);
if(MC_ReadActualPosition_0.Valid == 1)
{
    BasicControl.Status.ActPosition = MC_ReadActualPosition_0.Position;
}

/******************** MC_READACTUALVELOCITY *********************/
MC_ReadActualVelocity_0.Enable = (!MC_ReadActualVelocity_0.Error);
MC_ReadActualVelocity_0.Axis = Axis1Obj;
MC_ReadActualVelocity(&MC_ReadActualVelocity_0);
if(MC_ReadActualVelocity_0.Valid == 1)
{
    BasicControl.Status.ActVelocity = MC_ReadActualVelocity_0.Velocity;
}

/************************ MC_READAXISERROR **********************/
MC_ReadAxisError_0.Enable = !MC_ReadAxisError_0.Error;
MC_ReadAxisError_0.Axis = Axis1Obj;
MC_ReadAxisError_0.DataAddress = (UDINT)&(BasicControl.Status.ErrorText);
MC_ReadAxisError_0.DataLength = sizeof(BasicControl.Status.ErrorText);
strcpy((void*)&MC_ReadAxisError_0.DataObjectName,"acp10etxen");
MC_ReadAxisError(&MC_ReadAxisError_0);

/**************** CHECK FOR GENERAL AXIS ERROR ******************/
    if ((MC_ReadAxisError_0.AxisErrorID != 0) && (MC_ReadAxisError_0.Valid == 1))
    {
        AxisStep = STATE_ERROR_AXIS;
    }
/***************** CHECK IF POWER SHOULD BE OFF *******************/
    else if ((BasicControl.Command.Power == 0) && (MC_ReadAxisError_0.Valid == 1))
    {
        if ((MC_ReadStatus_0.Errorstop == 1) && (MC_ReadStatus_0.Valid == 1))
        {
            AxisStep = STATE_ERROR_RESET;
        }
        else
        {
            AxisStep = STATE_WAIT;
        }
    }

/* central monitoring of stop command attains a shorter reaction time in case of emergency stop */
/******************CHECK for STOP COMMAND************************/
    if (BasicControl.Command.Stop == 1)
    {
        if ((AxisStep >= STATE_HOME) && (AxisStep <= STATE_ERROR))
        {
            /* reset all FB execute inputs we use */
            MC_Home_0.Execute = 0;
            MC_Stop_0.Execute = 0;
            MC_MoveAbsolute_0.Execute = 0;
            MC_MoveAdditive_0.Execute = 0;
            MC_MoveVelocity_0.Execute = 0;
            MC_Halt_0.Execute = 0;
            MC_ReadAxisError_0.Acknowledge = 0;
            MC_Reset_0.Execute = 0;

            /* reset user commands */
            BasicControl.Command.Halt = 0;
            BasicControl.Command.Home = 0;
            BasicControl.Command.MoveJogPos = 0;
            BasicControl.Command.MoveJogNeg = 0;
            BasicControl.Command.MoveVelocity = 0;
            BasicControl.Command.MoveAbsolute = 0;
            BasicControl.Command.MoveAdditive = 0;
            AxisStep = STATE_STOP;
        }
    }

switch(AxisStep)
{
/******************** WAIT *************************/
    case STATE_WAIT:  /* STATE: Wait */
        if (BasicControl.Command.Power == 1)
        {
            AxisStep = STATE_POWER_ON;
        }
        else
        {
            MC_Power_0.Enable = 0;
        }

        /* reset all FB execute inputs we use */
        MC_Home_0.Execute = 0;
        MC_Stop_0.Execute = 0;
        MC_MoveAbsolute_0.Execute = 0;
        MC_MoveAdditive_0.Execute = 0;
        MC_MoveVelocity_0.Execute = 0;
        MC_Halt_0.Execute = 0;
        MC_ReadAxisError_0.Acknowledge = 0;
        MC_Reset_0.Execute = 0;

        /* reset user commands */
        BasicControl.Command.Halt = 0;
        BasicControl.Command.Home = 0;
        BasicControl.Command.MoveJogPos = 0;
        BasicControl.Command.MoveJogNeg = 0;
        BasicControl.Command.MoveVelocity = 0;
        BasicControl.Command.MoveAbsolute = 0;
        BasicControl.Command.MoveAdditive = 0;

        BasicControl.Status.ErrorID = 0;
    break;

/******************** POWER ON **********************/
    case STATE_POWER_ON:  /* STATE: Power on */
        MC_Power_0.Enable = 1;
        if (MC_Power_0.Status == 1)
        {
            AxisStep = STATE_READY;
        }
        /* if a power error occured go to error state */
        if (MC_Power_0.Error == 1)
        {
            BasicControl.Status.ErrorID = MC_Power_0.ErrorID;
            AxisStep = STATE_ERROR;
        }
    break;

/******************** READY **********************/
    case STATE_READY:  /* STATE: Waiting for commands */
        if (BasicControl.Command.Home == 1)
        {
            BasicControl.Command.Home = 0;
            AxisStep = STATE_HOME;
        }
        else if (BasicControl.Command.Stop == 1)
        {
            AxisStep = STATE_STOP;
        }
        else if (BasicControl.Command.MoveJogPos == 1)
        {
            AxisStep = STATE_JOG_POSITIVE;
        }
        else if (BasicControl.Command.MoveJogNeg == 1)
        {
            AxisStep = STATE_JOG_NEGATIVE;
        }
        else if (BasicControl.Command.MoveAbsolute == 1)
        {
            BasicControl.Command.MoveAbsolute = 0;
            AxisStep = STATE_MOVE_ABSOLUTE;
        }
        else if (BasicControl.Command.MoveAdditive == 1)
        {
            BasicControl.Command.MoveAdditive = 0;
            AxisStep = STATE_MOVE_ADDITIVE;
        }
        else if (BasicControl.Command.MoveVelocity == 1)
        {
            BasicControl.Command.MoveVelocity = 0;
            AxisStep = STATE_MOVE_VELOCITY;
        }
        else if (BasicControl.Command.Halt == 1)
        {
            BasicControl.Command.Halt = 0;
            AxisStep = STATE_HALT;
        }
    break;

/******************** HOME **********************/
    case STATE_HOME:  /* STATE: start homing process */
        MC_Home_0.Position = BasicControl.Parameter.HomePosition;
        MC_Home_0.HomingMode = BasicControl.Parameter.HomeMode;
        MC_Home_0.Execute = 1;
        if (MC_Home_0.Done == 1)
        {
            MC_Home_0.Execute = 0;
            AxisStep = STATE_READY;
        }
        /* if a homing error occured go to error state */
        if (MC_Home_0.Error == 1)
        {
            MC_Home_0.Execute = 0;
            BasicControl.Status.ErrorID = MC_Home_0.ErrorID;
            AxisStep = STATE_ERROR;
        }
    break;

/************************HALT MOVEMENT**************************/
    case STATE_HALT:  /* STATE: Stop the active movement */
        MC_Halt_0.Deceleration = BasicControl.Parameter.Deceleration;
        MC_Halt_0.Execute = 1;
        if (MC_Halt_0.Done == 1)
        {
            MC_Halt_0.Execute = 0;
            AxisStep = STATE_READY;
        }
        /*check if error occured */
        if (MC_Halt_0.Error == 1)
        {
            MC_Halt_0.Execute = 0;
            BasicControl.Status.ErrorID = MC_Halt_0.ErrorID;
            AxisStep = STATE_ERROR;
        }
    break;

/*********************** STOP MOVEMENT *************************/
    case STATE_STOP: /* STATE: Stop movement as long as command is set */
        MC_Stop_0.Deceleration = BasicControl.Parameter.Deceleration;
        MC_Stop_0.Execute = 1;
        /* if axis is stopped go to ready state */
        if ((MC_Stop_0.Done == 1) && (BasicControl.Command.Stop == 0))
        {
            MC_Stop_0.Execute = 0;
            AxisStep = STATE_READY;
        }
        /* check if error occured */
        if (MC_Stop_0.Error == 1)
        {
            BasicControl.Status.ErrorID = MC_Stop_0.ErrorID;
            MC_Stop_0.Execute = 0;
            AxisStep = STATE_ERROR;
        }
    break;

/******************** START JOG MOVEMENT POSITVE **********************/
    case STATE_JOG_POSITIVE:  /* STATE: Start jog movement in positive direction */
        MC_MoveVelocity_0.Velocity      = BasicControl.Parameter.JogVelocity;
        MC_MoveVelocity_0.Acceleration  = BasicControl.Parameter.Acceleration;
        MC_MoveVelocity_0.Deceleration  = BasicControl.Parameter.Deceleration;
        MC_MoveVelocity_0.Direction     = mcPOSITIVE_DIR;
        MC_MoveVelocity_0.Execute = 1;
        /* check if jog movement should be stopped */
        if (BasicControl.Command.MoveJogPos == 0)
        {
            MC_MoveVelocity_0.Execute = 0;
            AxisStep = STATE_HALT;
        }
        /* check if error occured */
        if (MC_MoveVelocity_0.Error == 1)
        {
            BasicControl.Status.ErrorID = MC_MoveVelocity_0.ErrorID;
            MC_MoveVelocity_0.Execute = 0;
            AxisStep = STATE_ERROR;
        }
    break;

/******************** START JOG MOVEMENT NEGATIVE **********************/
    case STATE_JOG_NEGATIVE:  /* STATE: Start jog movement in negative direction */
        MC_MoveVelocity_0.Velocity      = BasicControl.Parameter.JogVelocity;
        MC_MoveVelocity_0.Acceleration  = BasicControl.Parameter.Acceleration;
        MC_MoveVelocity_0.Deceleration  = BasicControl.Parameter.Deceleration;
        MC_MoveVelocity_0.Direction     = mcNEGATIVE_DIR;
        MC_MoveVelocity_0.Execute = 1;
        /* check if jog movement should be stopped */
        if (BasicControl.Command.MoveJogNeg == 0)
        {
            MC_MoveVelocity_0.Execute = 0;
            AxisStep = STATE_HALT;
        }
        /* check if error occured */
        if (MC_MoveVelocity_0.Error == 1)
        {
            BasicControl.Status.ErrorID = MC_MoveVelocity_0.ErrorID;
            MC_MoveVelocity_0.Execute = 0;
            AxisStep = STATE_ERROR;
        }
    break;

/******************** START ABSOLUTE MOVEMENT **********************/
    case STATE_MOVE_ABSOLUTE:  /* STATE: Start absolute movement */
        MC_MoveAbsolute_0.Position      = BasicControl.Parameter.Position;
        MC_MoveAbsolute_0.Velocity      = BasicControl.Parameter.Velocity;
        MC_MoveAbsolute_0.Acceleration  = BasicControl.Parameter.Acceleration;
        MC_MoveAbsolute_0.Deceleration  = BasicControl.Parameter.Deceleration;
        MC_MoveAbsolute_0.Direction     = BasicControl.Parameter.Direction;
        MC_MoveAbsolute_0.Execute = 1;
        /* check if commanded position is reached */
        if (BasicControl.Command.Halt == 1)
        {
            BasicControl.Command.Halt = 0;
            MC_MoveAbsolute_0.Execute = 0;
            AxisStep = STATE_HALT;
        }
        else if (MC_MoveAbsolute_0.Done == 1)
        {
            MC_MoveAbsolute_0.Execute = 0;
             AxisStep = STATE_READY;
        }
        /* check if error occured */
        if (MC_MoveAbsolute_0.Error == 1)
        {
            BasicControl.Status.ErrorID = MC_MoveAbsolute_0.ErrorID;
            MC_MoveAbsolute_0.Execute = 0;
            AxisStep = STATE_ERROR;
        }
    break;

/******************** START ADDITIVE MOVEMENT **********************/
    case STATE_MOVE_ADDITIVE:  /* STATE: Start additive movement */
        MC_MoveAdditive_0.Distance      = BasicControl.Parameter.Distance;
        MC_MoveAdditive_0.Velocity      = BasicControl.Parameter.Velocity;
        MC_MoveAdditive_0.Acceleration  = BasicControl.Parameter.Acceleration;
        MC_MoveAdditive_0.Deceleration  = BasicControl.Parameter.Deceleration;
        MC_MoveAdditive_0.Execute = 1;
        /* check if commanded distance is reached */
        if (BasicControl.Command.Halt == 1)
        {
            BasicControl.Command.Halt = 0;
            MC_MoveAdditive_0.Execute = 0;
            AxisStep = STATE_HALT;
        }
        else if (MC_MoveAdditive_0.Done == 1)
        {
            MC_MoveAdditive_0.Execute = 0;
             AxisStep = STATE_READY;
        }
        /* check if error occured */
        if (MC_MoveAdditive_0.Error == 1)
        {
            BasicControl.Status.ErrorID = MC_MoveAdditive_0.ErrorID;
            MC_MoveAdditive_0.Execute = 0;
            AxisStep = STATE_ERROR;
        }
    break;

/******************** START VELOCITY MOVEMENT **********************/
    case STATE_MOVE_VELOCITY:  /* STATE: Start velocity movement */
        MC_MoveVelocity_0.Velocity      = BasicControl.Parameter.Velocity;
        MC_MoveVelocity_0.Acceleration  = BasicControl.Parameter.Acceleration;
        MC_MoveVelocity_0.Deceleration  = BasicControl.Parameter.Deceleration;
        MC_MoveVelocity_0.Direction     = BasicControl.Parameter.Direction;
        MC_MoveVelocity_0.Execute = 1;
        /* check if commanded velocity is reached */
        if (BasicControl.Command.Halt == 1)
        {
            BasicControl.Command.Halt = 0;
            MC_MoveVelocity_0.Execute = 0;
            AxisStep = STATE_HALT;
        }
        else if (MC_MoveVelocity_0.InVelocity == 1)
        {
            MC_MoveVelocity_0.Execute = 0;
             AxisStep = STATE_READY;
        }
        /* check if error occured */
        if (MC_MoveVelocity_0.Error == 1)
        {
            BasicControl.Status.ErrorID = MC_MoveVelocity_0.ErrorID;
            MC_MoveVelocity_0.Execute = 0;
            AxisStep = STATE_ERROR;
        }
    break;

/******************** FB-ERROR OCCURED *************************/
    case STATE_ERROR:  /* STATE: Error */
        /* check if FB indicates an axis error */
        if (MC_ReadAxisError_0.AxisErrorCount != 0)
        {
            AxisStep = STATE_ERROR_AXIS;
        }
        else
        {
            if (BasicControl.Command.ErrorAcknowledge == 1)
            {
                BasicControl.Command.ErrorAcknowledge = 0;
                BasicControl.Status.ErrorID = 0;
                /* reset axis if it is in axis state ErrorStop */
                if ((MC_ReadStatus_0.Errorstop == 1) && (MC_ReadStatus_0.Valid == 1))
                {
                    AxisStep = STATE_ERROR_RESET;
                }
                else
                {
                    AxisStep = STATE_WAIT;
                }
            }
        }
    break;

/******************** AXIS-ERROR OCCURED *************************/
    case STATE_ERROR_AXIS:  /* STATE: Axis Error */
        if (MC_ReadAxisError_0.Valid == 1)
        {
            if (MC_ReadAxisError_0.AxisErrorID != 0)
            {
                BasicControl.Status.ErrorID = MC_ReadAxisError_0.AxisErrorID;
            }
            MC_ReadAxisError_0.Acknowledge = 0;
            if (BasicControl.Command.ErrorAcknowledge == 1)
            {
                BasicControl.Command.ErrorAcknowledge = 0;
                /* acknowledge axis error */
                if (MC_ReadAxisError_0.AxisErrorID != 0)
                {
                    MC_ReadAxisError_0.Acknowledge = 1;
                }
            }
            if (MC_ReadAxisError_0.AxisErrorCount == 0)
            {
                BasicControl.Status.ErrorID = 0;
                /* reset axis if it is in axis state ErrorStop */
                if ((MC_ReadStatus_0.Errorstop == 1) && (MC_ReadStatus_0.Valid == 1))
                {
                    AxisStep = STATE_ERROR_RESET;
                }
                else
                {
                    AxisStep = STATE_WAIT;
                }
            }
        }
    break;

/******************** RESET DONE *************************/
    case STATE_ERROR_RESET:  /* STATE: Wait for reset done */
        MC_Reset_0.Execute = 1;
        /* reset MC_Power.Enable if this FB is in Error*/
        if(MC_Power_0.Error == 1)
        {
            MC_Power_0.Enable = 0;
        }
        if(MC_Reset_0.Done == 1)
        {
            MC_Reset_0.Execute = 0;
            AxisStep = STATE_WAIT;
        }
        else if (MC_Reset_0.Error == 1)
        {
            MC_Reset_0.Execute = 0;
            AxisStep = STATE_ERROR;
        }
    break;

/******************** SEQUENCE END *************************/
}

/***************************************************************
        Function Block Calls
***************************************************************/

/************************** MC_POWER ****************************/
MC_Power_0.Axis = Axis1Obj;  /* pointer to axis */
MC_Power(&MC_Power_0);

/************************** MC_HOME *****************************/
MC_Home_0.Axis = Axis1Obj;
MC_Home(&MC_Home_0);

/********************** MC_MOVEABSOLUTE *************************/
MC_MoveAbsolute_0.Axis = Axis1Obj;
MC_MoveAbsolute(&MC_MoveAbsolute_0);

/********************** MC_MOVEADDITIVE *************************/
MC_MoveAdditive_0.Axis = Axis1Obj;
MC_MoveAdditive(&MC_MoveAdditive_0);

/********************** MC_MOVEVELOCITY *************************/
MC_MoveVelocity_0.Axis = Axis1Obj;
MC_MoveVelocity(&MC_MoveVelocity_0);

/************************** MC_STOP *****************************/
MC_Stop_0.Axis = Axis1Obj;
MC_Stop(&MC_Stop_0);

/**************************MC_HALT*******************************/
MC_Halt_0.Axis = Axis1Obj;
MC_Halt(&MC_Halt_0);

/************************** MC_RESET ****************************/
MC_Reset_0.Axis = Axis1Obj;
MC_Reset(&MC_Reset_0);

}
```

### Program Logical/Motion

#### Types.typ
```iecst
TYPE
	DistanceSensorInputsStruct : 	STRUCT
		LeftLSB : USINT;
		LeftMSB : USINT;
		MiddleLSB : USINT;
		MiddleMSB : USINT;
		RightLSB : USINT;
		RightMSB : USINT;
	END_STRUCT;
	InclineSensorInputsStruct : 	STRUCT
		MSB : USINT;
		LSB : USINT;
	END_STRUCT;
END_TYPE
```

#### Variables.var
```iecst
VAR
	DistanceSensorLeft : INT;
	DistanceSensorRight : INT;
	DistanceSensorMiddle : INT;
	DistanceSensorInputsVar : DistanceSensorInputsStruct;
	FieldAngle : REAL;
	InclineSensorInputsVar : InclineSensorInputsStruct;
END_VAR
```

#### variables.h
```c
#ifndef VARIABLES_H
#define VARIABLES_H

#include <bur/plctypes.h>
#include <bur/plc.h>  // evt nodig voor BOOL, etc.

extern BOOL i_HMI_Button_1;
extern BOOL i_HMI_Button_2;
extern BOOL i_HMI_Button_3;

extern BOOL o_HMI_Button_1;
extern BOOL o_HMI_Button_2;
extern BOOL o_HMI_Button_3;

#endif
```

#### Cyclic.cpp
```cpp
#include <bur/plctypes.h>
#include "variables.h"
#ifdef _DEFAULT_INCLUDES
	#include <AsDefault.h>
#endif

// amount of memory to be allocated for heap storage must be specified for every ANSI C++ program with the bur_heap_size variable
unsigned long bur_heap_size = 0xFFFF;

void _CYCLIC ProgramCyclic(void)
{
	INT distLeft = DistanceSensor(DistanceSensorInputsVar.LeftMSB, DistanceSensorInputsVar.LeftLSB);
	INT distMiddle = DistanceSensor(DistanceSensorInputsVar.MiddleMSB, DistanceSensorInputsVar.MiddleLSB);
	INT distRight = DistanceSensor(DistanceSensorInputsVar.RightMSB, DistanceSensorInputsVar.RightLSB);

	DistanceSensorLeft = (distLeft >= 30 && distLeft <= 300) ? distLeft : DistanceSensorLeft;
	DistanceSensorMiddle = (distMiddle >= 30 && distMiddle <= 300) ? distMiddle : DistanceSensorMiddle;
	DistanceSensorRight = (distRight >= 30 && distRight <= 300) ? distRight : DistanceSensorRight;
}
```

#### Init.cpp
```cpp
#include <bur/plctypes.h>

#ifdef _DEFAULT_INCLUDES
	#include <AsDefault.h>
#endif

void _INIT ProgramInit(void)
{
	// Insert code here
	bool i_HMI_Button_1;
	bool i_HMI_Button_2;
	bool i_HMI_Button_3;
	bool o_HMI_Button_1;
	bool o_HMI_Button_2;
	bool o_HMI_Button_3;
}
```

### Library Logical/Timer_CPP/Timer (ANSIC) - Object oriented IEC Timer
Depends on: standard

#### IECTonTimer.hpp
```cpp
/********************************************************************
 * COPYRIGHT --
 ********************************************************************
 * Library: Timer
 * File: IECTonTimer.hpp
 *******************************************************************/
#pragma once

#include <standard.h>
#include "ITimer.hpp"

/* The class IECTonTimer wraps a B&R TON function block.*/
class IECTonTimer : public ITimer
{
	private:
		TON_typ fubTON;

	public:
		IECTonTimer();
		IECTonTimer(signed long time);
		virtual ~IECTonTimer() {};
		virtual void start(bool start = 1);
		virtual void reset(bool reset = 0);
		virtual bool output();
		virtual void setTime(signed long time);
		virtual signed long getElapsedTime();

		virtual void cyclic();
};
```

#### IECTofTimer.hpp
```cpp
/********************************************************************
 * COPYRIGHT --
 ********************************************************************
 * Library: Timer
 * File: IECTonTimer.hpp
 *******************************************************************/
#pragma once

#include <standard.h>
#include "ITimer.hpp"

/* The class IECTonTimer wraps a B&R TOF function block.*/
class IECTofTimer : public ITimer
{
	private:
		TOF_typ fubTOF;

	public:
		IECTofTimer();
		IECTofTimer(signed long time);
		virtual ~IECTofTimer() {};
		virtual void start(bool start = 1);
		virtual void reset(bool reset = 1);
		virtual bool output();
		virtual void setTime(signed long time);
		virtual signed long getElapsedTime();

		virtual void cyclic();
};
```

#### IECTpTimer.cpp
```cpp
/********************************************************************
 * COPYRIGHT --
 ********************************************************************
 * Library: Timer
 * File: IECTpTimer.cpp
 *******************************************************************/

#include <string.h>
#include "IECTpTimer.hpp"

IECTpTimer::IECTpTimer()
{
	memset(&fubTP,0,sizeof(fubTP));
}

IECTpTimer::IECTpTimer(signed long time)
{
	memset(&fubTP,0,sizeof(fubTP));
	this->setTime(time);
}

void IECTpTimer::start(bool start)
{
	this->fubTP.IN = start;
}

void IECTpTimer::reset(bool reset)
{
	this->fubTP.IN = !reset;
}

void IECTpTimer::setTime(signed long time)
{
	this->fubTP.PT = time;
}

bool IECTpTimer::output()
{
	return this->fubTP.Q;
}

signed long IECTpTimer::getElapsedTime()
{
	return this->fubTP.ET;
}

/* This method has to be called cyclically in programms.*/
void IECTpTimer::cyclic()
{
	TP(&fubTP);
}
```

### Program Logical/Timer_CPP/TonTimer (ANSIC) - TON Sample
